  Call Extruder(256.15201)
  MoveL 1325 to (239.22, 155.88, 31.63) mm, rotated rx -180 ry 0 rz 180 deg; joints [-63.058, 52.64, -67.408, 63.827, 96.632, 13.225]
  MoveL 1326 to (239.22, 155.88, 31.63) mm, rotated rx -180 ry 0 rz 180 deg; joints [-63.058, 52.64, -67.408, 63.827, 96.632, 13.225]
  Call Extruder(256.33510)
  MoveL 1327 to (239.11, 156.17, 31.63) mm, rotated rx -180 ry 0 rz 180 deg; joints [-63.136, 52.655, -67.4, 63.902, 96.604, 13.213]
  MoveL 1328 to (239.11, 156.17, 31.63) mm, rotated rx -180 ry 0 rz 180 deg; joints [-63.136, 52.655, -67.4, 63.902, 96.604, 13.213]
  Call Extruder(256.49281)
  MoveL 1329 to (239, 156.42, 31.63) mm, rotated rx -180 ry 0 rz 180 deg; joints [-63.204, 52.668, -67.393, 63.966, 96.58, 13.203]
  MoveL 1330 to (239, 156.42, 31.63) mm, rotated rx -180 ry 0 rz 180 deg; joints [-63.204, 52.668, -67.393, 63.966, 96.58, 13.203]
  Call Extruder(256.65113)
  MoveL 1331 to (238.89, 156.67, 31.63) mm, rotated rx 180 ry 0 rz 180 deg; joints [-63.272, 52.68, -67.387, 64.031, 96.556, 13.193]
  MoveL 1332 to (238.89, 156.67, 31.63) mm, rotated rx 180 ry 0 rz 180 deg; joints [-63.272, 52.68, -67.387, 64.031, 96.556, 13.193]
  Call Extruder(256.83316)
  MoveL 1333 to (238.75, 156.94, 31.63) mm, rotated rx -180 ry 0 rz -180 deg; joints [-63.354, 52.694, -67.379, 64.109, 96.528, 13.183]
  MoveL 1334 to (238.75, 156.94, 31.63) mm, rotated rx -180 ry 0 rz -180 deg; joints [-63.354, 52.694, -67.379, 64.109, 96.528, 13.183]
  Call Extruder(257.03972)
  MoveL 1335 to (238.57, 157.25, 31.63) mm, rotated rx -180 ry 0 rz 180 deg; joints [-63.449, 52.708, -67.372, 64.2, 96.497, 13.174]
  MoveL 1336 to (238.57, 157.25, 31.63) mm, rotated rx -180 ry 0 rz 180 deg; joints [-63.449, 52.708, -67.372, 64.2, 96.497, 13.174]
  Call Extruder(257.24706)
  MoveL 1337 to (238.4, 157.55, 31.63) mm, rotated rx 180 ry 0 rz 180 deg; joints [-63.544, 52.722, -67.364, 64.291, 96.466, 13.165]
  MoveL 1338 to (238.4, 157.55, 31.63) mm, rotated rx 180 ry 0 rz 180 deg; joints [-63.544, 52.722, -67.364, 64.291, 96.466, 13.165]
  Call Extruder(257.45518)
  MoveL 1339 to (238.22, 157.85, 31.63) mm, rotated rx -180 ry 0 rz 180 deg; joints [-63.64, 52.736, -67.357, 64.383, 96.435, 13.156]
  MoveL 1340 to (238.22, 157.85, 31.63) mm, rotated rx -180 ry 0 rz 180 deg; joints [-63.64, 52.736, -67.357, 64.383, 96.435, 13.156]
  Call Extruder(257.57289)
  MoveL 1341 to (238.12, 158.02, 31.63) mm, rotated rx 180 ry 0 rz 180 deg; joints [-63.693, 52.744, -67.353, 64.434, 96.418, 13.151]
  MoveL 1342 to (238.12, 158.02, 31.63) mm, rotated rx 180 ry 0 rz 180 deg; joints [-63.693, 52.744, -67.353, 64.434, 96.418, 13.151]
  Call Extruder(257.90571)
  MoveL 1343 to (237.79, 158.48, 31.63) mm, rotated rx 180 ry 0 rz 180 deg; joints [-63.854, 52.763, -67.342, 64.588, 96.369, 13.142]
  MoveL 1344 to (237.79, 158.48, 31.63) mm, rotated rx 180 ry 0 rz 180 deg; joints [-63.854, 52.763, -67.342, 64.588, 96.369, 13.142]
  Call Extruder(258.23971)
  MoveL 1345 to (237.47, 158.93, 31.63) mm, rotated rx -180 ry 0 rz 180 deg; joints [-64.014, 52.782, -67.332, 64.742, 96.32, 13.133]
  MoveL 1346 to (237.47, 158.93, 31.63) mm, rotated rx -180 ry 0 rz 180 deg; joints [-64.014, 52.782, -67.332, 64.742, 96.32, 13.133]
  Call Extruder(258.40729)
  MoveL 1347 to (237.3, 159.15, 31.63) mm, rotated rx 180 ry 0 rz 180 deg; joints [-64.094, 52.792, -67.327, 64.819, 96.295, 13.128]
  Call Extruder(259.23663)
  MoveL 1348 to (236.39, 160.19, 31.63) mm, rotated rx -180 ry 0 rz 180 deg; joints [-64.505, 52.831, -67.306, 65.216, 96.177, 13.117]
  Call Extruder(259.86767)
  MoveL 1349 to (235.61, 160.89, 31.63) mm, rotated rx 180 ry 0 rz 180 deg; joints [-64.83, 52.852, -67.294, 65.531, 96.089, 13.121]
  MoveL 1350 to (235.61, 160.89, 31.63) mm, rotated rx 180 ry 0 rz 180 deg; joints [-64.83, 52.852, -67.294, 65.531, 96.089, 13.121]
  Call Extruder(260.06527)
  MoveL 1351 to (235.35, 161.1, 31.63) mm, rotated rx 180 ry 0 rz -180 deg; joints [-64.933, 52.858, -67.291, 65.631, 96.062, 13.123]
  Call Extruder(260.39930)
  MoveL 1352 to (234.9, 161.43, 31.63) mm, rotated rx -180 ry 0 rz -180 deg; joints [-65.109, 52.866, -67.287, 65.802, 96.017, 13.13]
  MoveL 1353 to (234.9, 161.43, 31.63) mm, rotated rx -180 ry 0 rz -180 deg; joints [-65.109, 52.866, -67.287, 65.802, 96.017, 13.13]
  Call Extruder(260.73214)
  MoveL 1354 to (234.45, 161.76, 31.63) mm, rotated rx -180 ry 0 rz -180 deg; joints [-65.285, 52.874, -67.282, 65.974, 95.972, 13.137]
  MoveL 1355 to (234.45, 161.76, 31.63) mm, rotated rx -180 ry 0 rz -180 deg; joints [-65.285, 52.874, -67.282, 65.974, 95.972, 13.137]
  Call Extruder(260.91134)
  MoveL 1356 to (234.21, 161.94, 31.63) mm, rotated rx 180 ry 0 rz -180 deg; joints [-65.381, 52.878, -67.28, 66.066, 95.947, 13.14]
  MoveL 1357 to (234.21, 161.94, 31.63) mm, rotated rx 180 ry 0 rz -180 deg; joints [-65.381, 52.878, -67.28, 66.066, 95.947, 13.14]
  Call Extruder(261.11946)
  MoveL 1358 to (233.9, 162.11, 31.63) mm, rotated rx 180 ry 0 rz -180 deg; joints [-65.493, 52.88, -67.279, 66.176, 95.92, 13.148]
  MoveL 1359 to (233.9, 162.11, 31.63) mm, rotated rx 180 ry 0 rz -180 deg; joints [-65.493, 52.88, -67.279, 66.176, 95.92, 13.148]
  Call Extruder(261.32679)
  MoveL 1360 to (233.6, 162.29, 31.63) mm, rotated rx -180 ry 0 rz 180 deg; joints [-65.605, 52.883, -67.277, 66.286, 95.893, 13.156]
  MoveL 1361 to (233.6, 162.29, 31.63) mm, rotated rx -180 ry 0 rz 180 deg; joints [-65.605, 52.883, -67.277, 66.286, 95.893, 13.156]
  Call Extruder(261.53335)
  MoveL 1362 to (233.29, 162.46, 31.63) mm, rotated rx 180 ry 0 rz 180 deg; joints [-65.718, 52.885, -67.276, 66.395, 95.866, 13.164]
  MoveL 1363 to (233.29, 162.46, 31.63) mm, rotated rx 180 ry 0 rz 180 deg; joints [-65.718, 52.885, -67.276, 66.395, 95.866, 13.164]
  Call Extruder(261.73913)
  MoveL 1364 to (232.99, 162.64, 31.63) mm, rotated rx -180 ry 0 rz 180 deg; joints [-65.83, 52.888, -67.275, 66.505, 95.839, 13.172]
  MoveL 1365 to (232.99, 162.64, 31.63) mm, rotated rx -180 ry 0 rz 180 deg; joints [-65.83, 52.888, -67.275, 66.505, 95.839, 13.172]
  Call Extruder(261.89741)
  MoveL 1366 to (232.74, 162.74, 31.63) mm, rotated rx -180 ry 0 rz 180 deg; joints [-65.917, 52.888, -67.275, 66.59, 95.819, 13.181]
  MoveL 1367 to (232.74, 162.74, 31.63) mm, rotated rx -180 ry 0 rz 180 deg; joints [-65.917, 52.888, -67.275, 66.59, 95.819, 13.181]
  Call Extruder(262.05508)
  MoveL 1368 to (232.49, 162.85, 31.63) mm, rotated rx -180 ry 0 rz 180 deg; joints [-66.004, 52.887, -67.275, 66.675, 95.8, 13.19]
  MoveL 1369 to (232.49, 162.85, 31.63) mm, rotated rx -180 ry 0 rz 180 deg; joints [-66.004, 52.887, -67.275, 66.675, 95.8, 13.19]
  Call Extruder(262.22517)
  MoveL 1370 to (232.22, 162.96, 31.63) mm, rotated rx 180 ry 0 rz 180 deg; joints [-66.099, 52.887, -67.275, 66.768, 95.778, 13.2]
  MoveL 1371 to (232.22, 162.96, 31.63) mm, rotated rx 180 ry 0 rz 180 deg; joints [-66.099, 52.887, -67.275, 66.768, 95.778, 13.2]
  Call Extruder(262.40753)
  MoveL 1372 to (231.93, 163.09, 31.63) mm, rotated rx -180 ry 0 rz 180 deg; joints [-66.2, 52.886, -67.275, 66.867, 95.755, 13.21]
  MoveL 1373 to (231.93, 163.09, 31.63) mm, rotated rx -180 ry 0 rz 180 deg; joints [-66.2, 52.886, -67.275, 66.867, 95.755, 13.21]
  Call Extruder(262.58914)
  MoveL 1374 to (231.64, 163.21, 31.63) mm, rotated rx -180 ry 0 rz 180 deg; joints [-66.302, 52.886, -67.276, 66.967, 95.733, 13.221]
  MoveL 1375 to (231.64, 163.21, 31.63) mm, rotated rx -180 ry 0 rz 180 deg; joints [-66.302, 52.886, -67.276, 66.967, 95.733, 13.221]
  Call Extruder(262.70258)
  MoveL 1376 to (231.45, 163.27, 31.63) mm, rotated rx -180 ry 0 rz -180 deg; joints [-66.365, 52.884, -67.277, 67.029, 95.719, 13.229]
  MoveL 1377 to (231.45, 163.27, 31.63) mm, rotated rx -180 ry 0 rz -180 deg; joints [-66.365, 52.884, -67.277, 67.029, 95.719, 13.229]
  Call Extruder(262.81558)
  MoveL 1378 to (231.26, 163.33, 31.63) mm, rotated rx 180 ry 0 rz -180 deg; joints [-66.428, 52.883, -67.277, 67.091, 95.705, 13.237]
  MoveL 1379 to (231.26, 163.33, 31.63) mm, rotated rx 180 ry 0 rz -180 deg; joints [-66.428, 52.883, -67.277, 67.091, 95.705, 13.237]
  Call Extruder(262.92814)
  MoveL 1380 to (231.07, 163.39, 31.63) mm, rotated rx 180 ry 0 rz 180 deg; joints [-66.492, 52.882, -67.278, 67.153, 95.692, 13.245]
  MoveL 1381 to (231.07, 163.39, 31.63) mm, rotated rx 180 ry 0 rz 180 deg; joints [-66.492, 52.882, -67.278, 67.153, 95.692, 13.245]
  Call Extruder(263.04025)
  MoveL 1382 to (230.88, 163.45, 31.63) mm, rotated rx 180 ry 0 rz 180 deg; joints [-66.555, 52.88, -67.279, 67.216, 95.678, 13.254]
  MoveL 1383 to (230.88, 163.45, 31.63) mm, rotated rx 180 ry 0 rz 180 deg; joints [-66.555, 52.88, -67.279, 67.216, 95.678, 13.254]
  Call Extruder(263.15191)
  MoveL 1384 to (230.69, 163.51, 31.63) mm, rotated rx 180 ry 0 rz -180 deg; joints [-66.619, 52.879, -67.28, 67.278, 95.664, 13.262]
  MoveL 1385 to (230.69, 163.51, 31.63) mm, rotated rx 180 ry 0 rz -180 deg; joints [-66.619, 52.879, -67.28, 67.278, 95.664, 13.262]
  Call Extruder(263.28301)
  MoveL 1386 to (230.47, 163.58, 31.63) mm, rotated rx -180 ry 0 rz 180 deg; joints [-66.694, 52.877, -67.281, 67.351, 95.648, 13.272]
  MoveL 1387 to (230.47, 163.58, 31.63) mm, rotated rx -180 ry 0 rz 180 deg; joints [-66.694, 52.877, -67.281, 67.351, 95.648, 13.272]
  Call Extruder(263.41354)
  MoveL 1388 to (230.25, 163.65, 31.63) mm, rotated rx -180 ry 0 rz 180 deg; joints [-66.768, 52.875, -67.282, 67.424, 95.632, 13.282]
  MoveL 1389 to (230.25, 163.65, 31.63) mm, rotated rx -180 ry 0 rz 180 deg; joints [-66.768, 52.875, -67.282, 67.424, 95.632, 13.282]
  Call Extruder(263.54350)
  MoveL 1390 to (230.02, 163.72, 31.63) mm, rotated rx 180 ry 0 rz -180 deg; joints [-66.843, 52.873, -67.283, 67.498, 95.616, 13.291]
  MoveL 1391 to (230.02, 163.72, 31.63) mm, rotated rx 180 ry 0 rz -180 deg; joints [-66.843, 52.873, -67.283, 67.498, 95.616, 13.291]
  Call Extruder(263.67290)
  MoveL 1392 to (229.8, 163.78, 31.63) mm, rotated rx 180 ry 0 rz -180 deg; joints [-66.918, 52.871, -67.284, 67.571, 95.6, 13.301]
  MoveL 1393 to (229.8, 163.78, 31.63) mm, rotated rx 180 ry 0 rz -180 deg; joints [-66.918, 52.871, -67.284, 67.571, 95.6, 13.301]
  Call Extruder(263.79488)
  MoveL 1394 to (229.59, 163.84, 31.63) mm, rotated rx -180 ry 0 rz 180 deg; joints [-66.988, 52.869, -67.285, 67.64, 95.585, 13.311]
  MoveL 1395 to (229.59, 163.84, 31.63) mm, rotated rx -180 ry 0 rz 180 deg; joints [-66.988, 52.869, -67.285, 67.64, 95.585, 13.311]
  Call Extruder(263.90973)
  MoveL 1396 to (229.38, 163.88, 31.63) mm, rotated rx 180 ry 0 rz 180 deg; joints [-67.054, 52.866, -67.287, 67.705, 95.572, 13.322]
  MoveL 1397 to (229.38, 163.88, 31.63) mm, rotated rx 180 ry 0 rz 180 deg; joints [-67.054, 52.866, -67.287, 67.705, 95.572, 13.322]
  Call Extruder(264.02412)
  MoveL 1398 to (229.18, 163.93, 31.63) mm, rotated rx 180 ry 0 rz -180 deg; joints [-67.12, 52.864, -67.288, 67.77, 95.558, 13.332]
  MoveL 1399 to (229.18, 163.93, 31.63) mm, rotated rx 180 ry 0 rz -180 deg; joints [-67.12, 52.864, -67.288, 67.77, 95.558, 13.332]
  Call Extruder(264.13806)
  MoveL 1400 to (228.97, 163.97, 31.63) mm, rotated rx -180 ry 0 rz 180 deg; joints [-67.187, 52.861, -67.29, 67.836, 95.544, 13.342]
  MoveL 1401 to (228.97, 163.97, 31.63) mm, rotated rx -180 ry 0 rz 180 deg; joints [-67.187, 52.861, -67.29, 67.836, 95.544, 13.342]
  Call Extruder(264.25155)
  MoveL 1402 to (228.77, 164.02, 31.63) mm, rotated rx 180 ry 0 rz 180 deg; joints [-67.253, 52.858, -67.291, 67.901, 95.531, 13.352]
  MoveL 1403 to (228.77, 164.02, 31.63) mm, rotated rx 180 ry 0 rz 180 deg; joints [-67.253, 52.858, -67.291, 67.901, 95.531, 13.352]
  Call Extruder(264.38884)
  MoveL 1404 to (228.52, 164.07, 31.63) mm, rotated rx 180 ry 0 rz 180 deg; joints [-67.333, 52.854, -67.293, 67.98, 95.514, 13.365]
  MoveL 1405 to (228.52, 164.07, 31.63) mm, rotated rx 180 ry 0 rz 180 deg; joints [-67.333, 52.854, -67.293, 67.98, 95.514, 13.365]
  Call Extruder(264.52551)
  MoveL 1406 to (228.27, 164.12, 31.63) mm, rotated rx 180 ry 0 rz -180 deg; joints [-67.413, 52.851, -67.295, 68.058, 95.498, 13.378]
  MoveL 1407 to (228.27, 164.12, 31.63) mm, rotated rx 180 ry 0 rz -180 deg; joints [-67.413, 52.851, -67.295, 68.058, 95.498, 13.378]
  Call Extruder(264.66157)
  MoveL 1408 to (228.02, 164.17, 31.63) mm, rotated rx 180 ry 0 rz 180 deg; joints [-67.494, 52.847, -67.297, 68.137, 95.481, 13.39]
  MoveL 1409 to (228.02, 164.17, 31.63) mm, rotated rx 180 ry 0 rz 180 deg; joints [-67.494, 52.847, -67.297, 68.137, 95.481, 13.39]
  Call Extruder(264.79703)
  MoveL 1410 to (227.77, 164.22, 31.63) mm, rotated rx 180 ry 0 rz -180 deg; joints [-67.574, 52.844, -67.299, 68.216, 95.465, 13.403]
  MoveL 1411 to (227.77, 164.22, 31.63) mm, rotated rx 180 ry 0 rz -180 deg; joints [-67.574, 52.844, -67.299, 68.216, 95.465, 13.403]
  Call Extruder(264.93187)
  MoveL 1412 to (227.52, 164.27, 31.63) mm, rotated rx -180 ry 0 rz -180 deg; joints [-67.654, 52.84, -67.301, 68.295, 95.448, 13.416]
  MoveL 1413 to (227.52, 164.27, 31.63) mm, rotated rx -180 ry 0 rz -180 deg; joints [-67.654, 52.84, -67.301, 68.295, 95.448, 13.416]
  Call Extruder(265.06610)
  MoveL 1414 to (227.27, 164.32, 31.63) mm, rotated rx 180 ry 0 rz -180 deg; joints [-67.735, 52.837, -67.303, 68.374, 95.431, 13.428]
  MoveL 1415 to (227.27, 164.32, 31.63) mm, rotated rx 180 ry 0 rz -180 deg; joints [-67.735, 52.837, -67.303, 68.374, 95.431, 13.428]
  Call Extruder(265.19972)
  MoveL 1416 to (227.03, 164.36, 31.63) mm, rotated rx -180 ry 0 rz 180 deg; joints [-67.815, 52.833, -67.305, 68.454, 95.415, 13.441]
  MoveL 1417 to (227.03, 164.36, 31.63) mm, rotated rx -180 ry 0 rz 180 deg; joints [-67.815, 52.833, -67.305, 68.454, 95.415, 13.441]
  Call Extruder(265.36183)
  MoveL 1418 to (226.72, 164.41, 31.63) mm, rotated rx -180 ry 0 rz 180 deg; joints [-67.912, 52.828, -67.307, 68.549, 95.395, 13.457]
  MoveL 1419 to (226.72, 164.41, 31.63) mm, rotated rx -180 ry 0 rz 180 deg; joints [-67.912, 52.828, -67.307, 68.549, 95.395, 13.457]
  Call Extruder(265.52320)
  MoveL 1420 to (226.41, 164.46, 31.63) mm, rotated rx -180 ry 0 rz 180 deg; joints [-68.01, 52.823, -67.31, 68.645, 95.375, 13.473]
  MoveL 1421 to (226.41, 164.46, 31.63) mm, rotated rx -180 ry 0 rz 180 deg; joints [-68.01, 52.823, -67.31, 68.645, 95.375, 13.473]
  Call Extruder(265.68385)
  MoveL 1422 to (226.11, 164.51, 31.63) mm, rotated rx -180 ry 0 rz -180 deg; joints [-68.107, 52.818, -67.313, 68.741, 95.355, 13.489]
  MoveL 1423 to (226.11, 164.51, 31.63) mm, rotated rx -180 ry 0 rz -180 deg; joints [-68.107, 52.818, -67.313, 68.741, 95.355, 13.489]
  Call Extruder(265.84377)
  MoveL 1424 to (225.8, 164.56, 31.63) mm, rotated rx -180 ry 0 rz -180 deg; joints [-68.205, 52.813, -67.316, 68.837, 95.335, 13.505]
  MoveL 1425 to (225.8, 164.56, 31.63) mm, rotated rx -180 ry 0 rz -180 deg; joints [-68.205, 52.813, -67.316, 68.837, 95.335, 13.505]
  Call Extruder(266.00296)
  MoveL 1426 to (225.5, 164.61, 31.63) mm, rotated rx -180 ry 0 rz -180 deg; joints [-68.303, 52.808, -67.318, 68.933, 95.315, 13.521]
  MoveL 1427 to (225.5, 164.61, 31.63) mm, rotated rx -180 ry 0 rz -180 deg; joints [-68.303, 52.808, -67.318, 68.933, 95.315, 13.521]
  Call Extruder(266.16143)
  MoveL 1428 to (225.19, 164.66, 31.63) mm, rotated rx -180 ry 0 rz 180 deg; joints [-68.4, 52.803, -67.321, 69.029, 95.295, 13.537]
  MoveL 1429 to (225.19, 164.66, 31.63) mm, rotated rx -180 ry 0 rz 180 deg; joints [-68.4, 52.803, -67.321, 69.029, 95.295, 13.537]
  Call Extruder(266.36030)
  MoveL 1430 to (224.8, 164.7, 31.63) mm, rotated rx -180 ry 0 rz 180 deg; joints [-68.522, 52.796, -67.325, 69.149, 95.27, 13.559]
  MoveL 1431 to (224.8, 164.7, 31.63) mm, rotated rx -180 ry 0 rz 180 deg; joints [-68.522, 52.796, -67.325, 69.149, 95.27, 13.559]
  Call Extruder(266.55831)
  MoveL 1432 to (224.42, 164.75, 31.63) mm, rotated rx 180 ry 0 rz 180 deg; joints [-68.645, 52.789, -67.329, 69.27, 95.245, 13.58]
  MoveL 1433 to (224.42, 164.75, 31.63) mm, rotated rx 180 ry 0 rz 180 deg; joints [-68.645, 52.789, -67.329, 69.27, 95.245, 13.58]
  Call Extruder(266.75545)
  MoveL 1434 to (224.03, 164.79, 31.63) mm, rotated rx 180 ry 0 rz 180 deg; joints [-68.767, 52.782, -67.333, 69.39, 95.221, 13.601]
  MoveL 1435 to (224.03, 164.79, 31.63) mm, rotated rx 180 ry 0 rz 180 deg; joints [-68.767, 52.782, -67.333, 69.39, 95.221, 13.601]
  Call Extruder(266.95173)
  MoveL 1436 to (223.64, 164.84, 31.63) mm, rotated rx 180 ry 0 rz -180 deg; joints [-68.89, 52.774, -67.336, 69.511, 95.196, 13.622]
  MoveL 1437 to (223.64, 164.84, 31.63) mm, rotated rx 180 ry 0 rz -180 deg; joints [-68.89, 52.774, -67.336, 69.511, 95.196, 13.622]
  Call Extruder(267.19740)
  MoveL 1438 to (223.15, 164.89, 31.63) mm, rotated rx 180 ry 0 rz 180 deg; joints [-69.043, 52.765, -67.342, 69.661, 95.165, 13.65]
  MoveL 1439 to (223.15, 164.89, 31.63) mm, rotated rx 180 ry 0 rz 180 deg; joints [-69.043, 52.765, -67.342, 69.661, 95.165, 13.65]
  Call Extruder(267.49209)
  MoveL 1440 to (222.56, 164.93, 31.63) mm, rotated rx 180 ry 0 rz 180 deg; joints [-69.227, 52.753, -67.348, 69.843, 95.128, 13.683]
  MoveL 1441 to (222.56, 164.93, 31.63) mm, rotated rx 180 ry 0 rz 180 deg; joints [-69.227, 52.753, -67.348, 69.843, 95.128, 13.683]
  Call Extruder(267.78545)
  MoveL 1442 to (221.97, 164.98, 31.63) mm, rotated rx 180 ry 0 rz 180 deg; joints [-69.411, 52.741, -67.354, 70.024, 95.09, 13.717]
  MoveL 1443 to (221.97, 164.98, 31.63) mm, rotated rx 180 ry 0 rz 180 deg; joints [-69.411, 52.741, -67.354, 70.024, 95.09, 13.717]
  Call Extruder(268.21876)
  MoveL 1444 to (221.1, 165.03, 31.63) mm, rotated rx 180 ry 0 rz -180 deg; joints [-69.684, 52.722, -67.365, 70.292, 95.035, 13.768]
  MoveL 1445 to (221.1, 165.03, 31.63) mm, rotated rx 180 ry 0 rz -180 deg; joints [-69.684, 52.722, -67.365, 70.292, 95.035, 13.768]
  Call Extruder(268.79092)
  MoveL 1446 to (219.94, 165.07, 31.63) mm, rotated rx -180 ry 0 rz 180 deg; joints [-70.044, 52.696, -67.379, 70.647, 94.963, 13.836]
  MoveL 1447 to (219.94, 165.07, 31.63) mm, rotated rx -180 ry 0 rz 180 deg; joints [-70.044, 52.696, -67.379, 70.647, 94.963, 13.836]
  Call Extruder(269.21879)
  MoveL 1448 to (219.06, 165.09, 31.63) mm, rotated rx -180 ry 0 rz 180 deg; joints [-70.315, 52.675, -67.389, 70.913, 94.908, 13.888]
  Call Extruder(385.86744)
  MoveL 1449 to (-19.06, 165.09, 31.63) mm, rotated rx -180 ry 0 rz 180 deg; joints [-137.325, 57.005, -63.843, 137.121, 84.978, 4.647]
  MoveL 1450 to (-19.06, 165.09, 31.63) mm, rotated rx -180 ry 0 rz 180 deg; joints [-137.325, 57.005, -63.843, 137.121, 84.978, 4.647]
  Call Extruder(386.58306)
  MoveL 1451 to (-20.52, 165.05, 31.63) mm, rotated rx 180 ry 0 rz -180 deg; joints [-137.563, 57.061, -63.774, 137.367, 85.05, 4.541]
  MoveL 1452 to (-20.52, 165.05, 31.63) mm, rotated rx 180 ry 0 rz -180 deg; joints [-137.563, 57.061, -63.774, 137.367, 85.05, 4.541]
  Call Extruder(387.15780)
  MoveL 1453 to (-21.68, 165, 31.63) mm, rotated rx -180 ry 0 rz -180 deg; joints [-137.754, 57.105, -63.719, 137.564, 85.108, 4.458]
  MoveL 1454 to (-21.68, 165, 31.63) mm, rotated rx -180 ry 0 rz -180 deg; joints [-137.754, 57.105, -63.719, 137.564, 85.108, 4.458]
  Call Extruder(387.45117)
  MoveL 1455 to (-22.27, 164.95, 31.63) mm, rotated rx 180 ry 0 rz 180 deg; joints [-137.855, 57.126, -63.692, 137.667, 85.136, 4.417]
  MoveL 1456 to (-22.27, 164.95, 31.63) mm, rotated rx 180 ry 0 rz 180 deg; joints [-137.855, 57.126, -63.692, 137.667, 85.136, 4.417]
  Call Extruder(387.74586)
  MoveL 1457 to (-22.86, 164.91, 31.63) mm, rotated rx 180 ry 0 rz -180 deg; joints [-137.955, 57.148, -63.665, 137.77, 85.165, 4.375]
  MoveL 1458 to (-22.86, 164.91, 31.63) mm, rotated rx 180 ry 0 rz -180 deg; joints [-137.955, 57.148, -63.665, 137.77, 85.165, 4.375]
  Call Extruder(388.04189)
  MoveL 1459 to (-23.45, 164.86, 31.63) mm, rotated rx -180 ry 0 rz -180 deg; joints [-138.054, 57.169, -63.638, 137.872, 85.193, 4.334]
  MoveL 1460 to (-23.45, 164.86, 31.63) mm, rotated rx -180 ry 0 rz -180 deg; joints [-138.054, 57.169, -63.638, 137.872, 85.193, 4.334]
  Call Extruder(388.23816)
  MoveL 1461 to (-23.83, 164.82, 31.63) mm, rotated rx -180 ry 0 rz 180 deg; joints [-138.122, 57.183, -63.621, 137.942, 85.211, 4.308]
  MoveL 1462 to (-23.83, 164.82, 31.63) mm, rotated rx -180 ry 0 rz 180 deg; joints [-138.122, 57.183, -63.621, 137.942, 85.211, 4.308]
  Call Extruder(388.43530)
  MoveL 1463 to (-24.22, 164.77, 31.63) mm, rotated rx 180 ry 0 rz 180 deg; joints [-138.19, 57.196, -63.604, 138.012, 85.229, 4.282]
  MoveL 1464 to (-24.22, 164.77, 31.63) mm, rotated rx 180 ry 0 rz 180 deg; joints [-138.19, 57.196, -63.604, 138.012, 85.229, 4.282]
  Call Extruder(388.63331)
  MoveL 1465 to (-24.61, 164.72, 31.63) mm, rotated rx -180 ry 0 rz -180 deg; joints [-138.258, 57.21, -63.586, 138.081, 85.246, 4.255]
  MoveL 1466 to (-24.61, 164.72, 31.63) mm, rotated rx -180 ry 0 rz -180 deg; joints [-138.258, 57.21, -63.586, 138.081, 85.246, 4.255]
  Call Extruder(388.83219)
  MoveL 1467 to (-25, 164.68, 31.63) mm, rotated rx -180 ry 0 rz 180 deg; joints [-138.325, 57.223, -63.569, 138.151, 85.265, 4.229]
  MoveL 1468 to (-25, 164.68, 31.63) mm, rotated rx -180 ry 0 rz 180 deg; joints [-138.325, 57.223, -63.569, 138.151, 85.265, 4.229]
  Call Extruder(389.01127)
  MoveL 1469 to (-25.34, 164.63, 31.63) mm, rotated rx 180 ry 0 rz 180 deg; joints [-138.387, 57.235, -63.554, 138.213, 85.28, 4.206]
  MoveL 1470 to (-25.34, 164.63, 31.63) mm, rotated rx 180 ry 0 rz 180 deg; joints [-138.387, 57.235, -63.554, 138.213, 85.28, 4.206]
  Call Extruder(389.17046)
  MoveL 1471 to (-25.65, 164.58, 31.63) mm, rotated rx -180 ry 0 rz 180 deg; joints [-138.442, 57.245, -63.54, 138.27, 85.294, 4.185]
  MoveL 1472 to (-25.65, 164.58, 31.63) mm, rotated rx -180 ry 0 rz 180 deg; joints [-138.442, 57.245, -63.54, 138.27, 85.294, 4.185]
  Call Extruder(389.33039)
  MoveL 1473 to (-25.96, 164.54, 31.63) mm, rotated rx 180 ry 0 rz -180 deg; joints [-138.497, 57.256, -63.527, 138.327, 85.307, 4.165]
  MoveL 1474 to (-25.96, 164.54, 31.63) mm, rotated rx 180 ry 0 rz -180 deg; joints [-138.497, 57.256, -63.527, 138.327, 85.307, 4.165]
  Call Extruder(389.49104)
  MoveL 1475 to (-26.26, 164.49, 31.63) mm, rotated rx 180 ry 0 rz 180 deg; joints [-138.552, 57.266, -63.514, 138.383, 85.321, 4.145]
  MoveL 1476 to (-26.26, 164.49, 31.63) mm, rotated rx 180 ry 0 rz 180 deg; joints [-138.552, 57.266, -63.514, 138.383, 85.321, 4.145]
  Call Extruder(389.65242)
  MoveL 1477 to (-26.57, 164.44, 31.63) mm, rotated rx -180 ry 0 rz 180 deg; joints [-138.607, 57.276, -63.5, 138.439, 85.335, 4.125]
  MoveL 1478 to (-26.57, 164.44, 31.63) mm, rotated rx -180 ry 0 rz 180 deg; joints [-138.607, 57.276, -63.5, 138.439, 85.335, 4.125]
  Call Extruder(389.81452)
  MoveL 1479 to (-26.87, 164.39, 31.63) mm, rotated rx -180 ry 0 rz 180 deg; joints [-138.662, 57.287, -63.487, 138.496, 85.348, 4.104]
  MoveL 1480 to (-26.87, 164.39, 31.63) mm, rotated rx -180 ry 0 rz 180 deg; joints [-138.662, 57.287, -63.487, 138.496, 85.348, 4.104]
  Call Extruder(389.96273)
  MoveL 1481 to (-27.15, 164.34, 31.63) mm, rotated rx 180 ry 0 rz -180 deg; joints [-138.713, 57.296, -63.475, 138.547, 85.361, 4.086]
  MoveL 1482 to (-27.15, 164.34, 31.63) mm, rotated rx 180 ry 0 rz -180 deg; joints [-138.713, 57.296, -63.475, 138.547, 85.361, 4.086]
  Call Extruder(390.09696)
  MoveL 1483 to (-27.4, 164.29, 31.63) mm, rotated rx -180 ry 0 rz 180 deg; joints [-138.759, 57.304, -63.465, 138.595, 85.371, 4.07]
  MoveL 1484 to (-27.4, 164.29, 31.63) mm, rotated rx -180 ry 0 rz 180 deg; joints [-138.759, 57.304, -63.465, 138.595, 85.371, 4.07]
  Call Extruder(390.23180)
  MoveL 1485 to (-27.65, 164.24, 31.63) mm, rotated rx -180 ry 0 rz 180 deg; joints [-138.806, 57.312, -63.454, 138.642, 85.382, 4.054]
  MoveL 1486 to (-27.65, 164.24, 31.63) mm, rotated rx -180 ry 0 rz 180 deg; joints [-138.806, 57.312, -63.454, 138.642, 85.382, 4.054]
  Call Extruder(390.36725)
  MoveL 1487 to (-27.9, 164.19, 31.63) mm, rotated rx -180 ry 0 rz 180 deg; joints [-138.852, 57.32, -63.444, 138.689, 85.392, 4.038]
  MoveL 1488 to (-27.9, 164.19, 31.63) mm, rotated rx -180 ry 0 rz 180 deg; joints [-138.852, 57.32, -63.444, 138.689, 85.392, 4.038]
  Call Extruder(390.50331)
  MoveL 1489 to (-28.15, 164.14, 31.63) mm, rotated rx -180 ry 0 rz 180 deg; joints [-138.898, 57.328, -63.433, 138.736, 85.403, 4.022]
  MoveL 1490 to (-28.15, 164.14, 31.63) mm, rotated rx -180 ry 0 rz 180 deg; joints [-138.898, 57.328, -63.433, 138.736, 85.403, 4.022]
  Call Extruder(390.63999)
  MoveL 1491 to (-28.4, 164.09, 31.63) mm, rotated rx 180 ry 0 rz 180 deg; joints [-138.944, 57.336, -63.422, 138.784, 85.414, 4.006]
  MoveL 1492 to (-28.4, 164.09, 31.63) mm, rotated rx 180 ry 0 rz 180 deg; joints [-138.944, 57.336, -63.422, 138.784, 85.414, 4.006]
  Call Extruder(390.77727)
  MoveL 1493 to (-28.65, 164.04, 31.63) mm, rotated rx -180 ry 0 rz 180 deg; joints [-138.99, 57.344, -63.412, 138.831, 85.425, 3.99]
  MoveL 1494 to (-28.65, 164.04, 31.63) mm, rotated rx -180 ry 0 rz 180 deg; joints [-138.99, 57.344, -63.412, 138.831, 85.425, 3.99]
  Call Extruder(390.90294)
  MoveL 1495 to (-28.87, 164, 31.63) mm, rotated rx -180 ry 0 rz -180 deg; joints [-139.032, 57.351, -63.402, 138.874, 85.434, 3.976]
  MoveL 1496 to (-28.87, 164, 31.63) mm, rotated rx -180 ry 0 rz -180 deg; joints [-139.032, 57.351, -63.402, 138.874, 85.434, 3.976]
  Call Extruder(391.01688)
  MoveL 1497 to (-29.08, 163.95, 31.63) mm, rotated rx -180 ry 0 rz 180 deg; joints [-139.071, 57.357, -63.394, 138.913, 85.443, 3.963]
  MoveL 1498 to (-29.08, 163.95, 31.63) mm, rotated rx -180 ry 0 rz 180 deg; joints [-139.071, 57.357, -63.394, 138.913, 85.443, 3.963]
  Call Extruder(391.13127)
  MoveL 1499 to (-29.28, 163.91, 31.63) mm, rotated rx -180 ry 0 rz -180 deg; joints [-139.109, 57.364, -63.385, 138.952, 85.452, 3.95]
  MoveL 1500 to (-29.28, 163.91, 31.63) mm, rotated rx -180 ry 0 rz -180 deg; joints [-139.109, 57.364, -63.385, 138.952, 85.452, 3.95]
  Call Extruder(391.24612)
  MoveL 1501 to (-29.48, 163.86, 31.63) mm, rotated rx 180 ry 0 rz 180 deg; joints [-139.147, 57.37, -63.377, 138.991, 85.46, 3.937]
  MoveL 1502 to (-29.48, 163.86, 31.63) mm, rotated rx 180 ry 0 rz 180 deg; joints [-139.147, 57.37, -63.377, 138.991, 85.46, 3.937]
  Call Extruder(391.36141)
  MoveL 1503 to (-29.69, 163.82, 31.63) mm, rotated rx -180 ry 0 rz -180 deg; joints [-139.186, 57.377, -63.368, 139.03, 85.469, 3.924]
  MoveL 1504 to (-29.69, 163.82, 31.63) mm, rotated rx -180 ry 0 rz -180 deg; joints [-139.186, 57.377, -63.368, 139.03, 85.469, 3.924]
  Call Extruder(391.49081)
  MoveL 1505 to (-29.91, 163.75, 31.63) mm, rotated rx -180 ry 0 rz -180 deg; joints [-139.231, 57.383, -63.359, 139.076, 85.477, 3.911]
  MoveL 1506 to (-29.91, 163.75, 31.63) mm, rotated rx -180 ry 0 rz -180 deg; joints [-139.231, 57.383, -63.359, 139.076, 85.477, 3.911]
  Call Extruder(391.62077)
  MoveL 1507 to (-30.14, 163.68, 31.63) mm, rotated rx 180 ry 0 rz 180 deg; joints [-139.276, 57.39, -63.351, 139.122, 85.486, 3.897]
  MoveL 1508 to (-30.14, 163.68, 31.63) mm, rotated rx 180 ry 0 rz 180 deg; joints [-139.276, 57.39, -63.351, 139.122, 85.486, 3.897]
  Call Extruder(391.75130)
  MoveL 1509 to (-30.36, 163.61, 31.63) mm, rotated rx -180 ry 0 rz 180 deg; joints [-139.321, 57.396, -63.342, 139.168, 85.494, 3.884]
  MoveL 1510 to (-30.36, 163.61, 31.63) mm, rotated rx -180 ry 0 rz 180 deg; joints [-139.321, 57.396, -63.342, 139.168, 85.494, 3.884]
  Call Extruder(391.88239)
  MoveL 1511 to (-30.58, 163.55, 31.63) mm, rotated rx -180 ry 0 rz 180 deg; joints [-139.366, 57.403, -63.334, 139.214, 85.502, 3.87]
  MoveL 1512 to (-30.58, 163.55, 31.63) mm, rotated rx -180 ry 0 rz 180 deg; joints [-139.366, 57.403, -63.334, 139.214, 85.502, 3.87]
  Call Extruder(392.00403)
  MoveL 1513 to (-30.79, 163.48, 31.63) mm, rotated rx -180 ry 0 rz 180 deg; joints [-139.408, 57.408, -63.326, 139.256, 85.51, 3.858]
  MoveL 1514 to (-30.79, 163.48, 31.63) mm, rotated rx -180 ry 0 rz 180 deg; joints [-139.408, 57.408, -63.326, 139.256, 85.51, 3.858]
  Call Extruder(392.11615)
  MoveL 1515 to (-30.98, 163.42, 31.63) mm, rotated rx -180 ry 0 rz -180 deg; joints [-139.446, 57.414, -63.319, 139.295, 85.517, 3.847]
  MoveL 1516 to (-30.98, 163.42, 31.63) mm, rotated rx -180 ry 0 rz -180 deg; joints [-139.446, 57.414, -63.319, 139.295, 85.517, 3.847]
  Call Extruder(392.22871)
  MoveL 1517 to (-31.17, 163.36, 31.63) mm, rotated rx -180 ry 0 rz -180 deg; joints [-139.485, 57.419, -63.311, 139.335, 85.524, 3.836]
  MoveL 1518 to (-31.17, 163.36, 31.63) mm, rotated rx -180 ry 0 rz -180 deg; joints [-139.485, 57.419, -63.311, 139.335, 85.524, 3.836]
  Call Extruder(392.34171)
  MoveL 1519 to (-31.35, 163.3, 31.63) mm, rotated rx -180 ry 0 rz 180 deg; joints [-139.523, 57.424, -63.304, 139.374, 85.531, 3.825]
  MoveL 1520 to (-31.35, 163.3, 31.63) mm, rotated rx -180 ry 0 rz 180 deg; joints [-139.523, 57.424, -63.304, 139.374, 85.531, 3.825]
  Call Extruder(392.45516)
  MoveL 1521 to (-31.54, 163.24, 31.63) mm, rotated rx 180 ry 0 rz -180 deg; joints [-139.562, 57.43, -63.297, 139.413, 85.537, 3.814]
  MoveL 1522 to (-31.54, 163.24, 31.63) mm, rotated rx 180 ry 0 rz -180 deg; joints [-139.562, 57.43, -63.297, 139.413, 85.537, 3.814]
  Call Extruder(392.60280)
  MoveL 1523 to (-31.78, 163.15, 31.63) mm, rotated rx -180 ry 0 rz 180 deg; joints [-139.613, 57.436, -63.289, 139.465, 85.545, 3.8]
  MoveL 1524 to (-31.78, 163.15, 31.63) mm, rotated rx -180 ry 0 rz 180 deg; joints [-139.613, 57.436, -63.289, 139.465, 85.545, 3.8]
  Call Extruder(392.78516)
  MoveL 1525 to (-32.08, 163.02, 31.63) mm, rotated rx 180 ry 0 rz 180 deg; joints [-139.677, 57.443, -63.279, 139.53, 85.554, 3.784]
  MoveL 1526 to (-32.08, 163.02, 31.63) mm, rotated rx 180 ry 0 rz 180 deg; joints [-139.677, 57.443, -63.279, 139.53, 85.554, 3.784]
  Call Extruder(392.96827)
  MoveL 1527 to (-32.37, 162.91, 31.63) mm, rotated rx -180 ry 0 rz -180 deg; joints [-139.741, 57.451, -63.269, 139.595, 85.563, 3.767]
  MoveL 1528 to (-32.37, 162.91, 31.63) mm, rotated rx -180 ry 0 rz -180 deg; joints [-139.741, 57.451, -63.269, 139.595, 85.563, 3.767]
  Call Extruder(393.12594)
  MoveL 1529 to (-32.62, 162.8, 31.63) mm, rotated rx 180 ry 0 rz 180 deg; joints [-139.796, 57.457, -63.26, 139.65, 85.571, 3.754]
  MoveL 1530 to (-32.62, 162.8, 31.63) mm, rotated rx 180 ry 0 rz 180 deg; joints [-139.796, 57.457, -63.26, 139.65, 85.571, 3.754]
  Call Extruder(393.28422)
  MoveL 1531 to (-32.86, 162.69, 31.63) mm, rotated rx 180 ry 0 rz 180 deg; joints [-139.851, 57.463, -63.252, 139.706, 85.578, 3.74]
  MoveL 1532 to (-32.86, 162.69, 31.63) mm, rotated rx 180 ry 0 rz 180 deg; joints [-139.851, 57.463, -63.252, 139.706, 85.578, 3.74]
  Call Extruder(393.46623)
  MoveL 1533 to (-33.14, 162.55, 31.63) mm, rotated rx -180 ry 0 rz 180 deg; joints [-139.916, 57.469, -63.244, 139.772, 85.585, 3.726]
  MoveL 1534 to (-33.14, 162.55, 31.63) mm, rotated rx -180 ry 0 rz 180 deg; joints [-139.916, 57.469, -63.244, 139.772, 85.585, 3.726]
  Call Extruder(393.67279)
  MoveL 1535 to (-33.45, 162.37, 31.63) mm, rotated rx -180 ry 0 rz -180 deg; joints [-139.991, 57.475, -63.235, 139.848, 85.591, 3.711]
  MoveL 1536 to (-33.45, 162.37, 31.63) mm, rotated rx -180 ry 0 rz -180 deg; joints [-139.991, 57.475, -63.235, 139.848, 85.591, 3.711]
  Call Extruder(393.88012)
  MoveL 1537 to (-33.75, 162.2, 31.63) mm, rotated rx 180 ry 0 rz -180 deg; joints [-140.065, 57.481, -63.227, 139.923, 85.597, 3.695]
  MoveL 1538 to (-33.75, 162.2, 31.63) mm, rotated rx 180 ry 0 rz -180 deg; joints [-140.065, 57.481, -63.227, 139.923, 85.597, 3.695]
  Call Extruder(394.08824)
  MoveL 1539 to (-34.05, 162.02, 31.63) mm, rotated rx 180 ry 0 rz 180 deg; joints [-140.14, 57.487, -63.219, 139.999, 85.604, 3.68]
  MoveL 1540 to (-34.05, 162.02, 31.63) mm, rotated rx 180 ry 0 rz 180 deg; joints [-140.14, 57.487, -63.219, 139.999, 85.604, 3.68]
  Call Extruder(394.20594)
  MoveL 1541 to (-34.23, 161.92, 31.63) mm, rotated rx 180 ry 0 rz 180 deg; joints [-140.182, 57.491, -63.214, 140.041, 85.607, 3.672]
  MoveL 1542 to (-34.23, 161.92, 31.63) mm, rotated rx 180 ry 0 rz 180 deg; joints [-140.182, 57.491, -63.214, 140.041, 85.607, 3.672]
  Call Extruder(394.53878)
  MoveL 1543 to (-34.68, 161.59, 31.63) mm, rotated rx 180 ry 0 rz 180 deg; joints [-140.305, 57.498, -63.204, 140.165, 85.612, 3.652]
  MoveL 1544 to (-34.68, 161.59, 31.63) mm, rotated rx 180 ry 0 rz 180 deg; joints [-140.305, 57.498, -63.204, 140.165, 85.612, 3.652]
  Call Extruder(394.87281)
  MoveL 1545 to (-35.13, 161.27, 31.63) mm, rotated rx -180 ry 0 rz 180 deg; joints [-140.427, 57.505, -63.195, 140.288, 85.617, 3.632]
  MoveL 1546 to (-35.13, 161.27, 31.63) mm, rotated rx -180 ry 0 rz 180 deg; joints [-140.427, 57.505, -63.195, 140.288, 85.617, 3.632]
  Call Extruder(395.04040)
  MoveL 1547 to (-35.35, 161.1, 31.63) mm, rotated rx 180 ry 0 rz 180 deg; joints [-140.489, 57.508, -63.19, 140.35, 85.62, 3.622]
  Call Extruder(395.86969)
  MoveL 1548 to (-36.39, 160.19, 31.63) mm, rotated rx 180 ry 0 rz 180 deg; joints [-140.797, 57.52, -63.174, 140.66, 85.621, 3.581]
  Call Extruder(396.50077)
  MoveL 1549 to (-37.09, 159.4, 31.63) mm, rotated rx -180 ry 0 rz -180 deg; joints [-141.034, 57.522, -63.171, 140.898, 85.611, 3.559]
  MoveL 1550 to (-37.09, 159.4, 31.63) mm, rotated rx -180 ry 0 rz -180 deg; joints [-141.034, 57.522, -63.171, 140.898, 85.611, 3.559]
  Call Extruder(396.69836)
  MoveL 1551 to (-37.3, 159.15, 31.63) mm, rotated rx -180 ry 0 rz 180 deg; joints [-141.109, 57.522, -63.17, 140.972, 85.607, 3.553]
  Call Extruder(397.03238)
  MoveL 1552 to (-37.63, 158.7, 31.63) mm, rotated rx -180 ry 0 rz 180 deg; joints [-141.235, 57.521, -63.172, 141.098, 85.596, 3.546]
  MoveL 1553 to (-37.63, 158.7, 31.63) mm, rotated rx -180 ry 0 rz 180 deg; joints [-141.235, 57.521, -63.172, 141.098, 85.596, 3.546]
  Call Extruder(397.26956)
  MoveL 1554 to (-37.87, 158.38, 31.63) mm, rotated rx 180 ry 0 rz 180 deg; joints [-141.324, 57.52, -63.174, 141.188, 85.589, 3.54]
  Set speed (130.0 mm/s)
  MoveL 1555 to (-39.5, 155.42, 31.63) mm, rotated rx -180 ry 0 rz -180 deg; joints [-142.08, 57.492, -63.212, 141.941, 85.491, 3.522]
  MoveL 1556 to (-39.51, 155.42, 41.04) mm, rotated rx -180 ry 0 rz 180 deg; joints [-142.08, 58.93, -65.352, 141.905, 84.938, 3.957]
  Call Extruder(395.26956)
  Set speed (40.0 mm/s)
  MoveL 1557 to (-39.51, 155.42, 41.04) mm, rotated rx -180 ry 0 rz 180 deg; joints [-142.08, 58.93, -65.352, 141.905, 84.938, 3.957]
  Call Extruder(0.00000)
  Set speed (130.0 mm/s)
  MoveL 1558 to (-39.41, 155.44, 41.04) mm, rotated rx -180 ry 0 rz 180 deg; joints [-142.064, 58.926, -65.356, 141.888, 84.932, 3.964]
  Call Extruder(2.00000)
  Set speed (40.0 mm/s)
  MoveL 1559 to (-39.41, 155.44, 41.04) mm, rotated rx -180 ry 0 rz 180 deg; joints [-142.064, 58.926, -65.356, 141.888, 84.932, 3.964]
  Set speed (30.0 mm/s)
  MoveL 1560 to (-39.41, 155.44, 41.04) mm, rotated rx -180 ry 0 rz 180 deg; joints [-142.064, 58.926, -65.356, 141.888, 84.932, 3.964]
  Call Extruder(2.05684)
  MoveL 1561 to (-39.44, 155.34, 41.04) mm, rotated rx -180 ry 0 rz 180 deg; joints [-142.085, 58.924, -65.359, 141.909, 84.928, 3.964]
  MoveL 1562 to (-39.44, 155.34, 41.04) mm, rotated rx -180 ry 0 rz 180 deg; joints [-142.085, 58.924, -65.359, 141.909, 84.928, 3.964]
  Call Extruder(2.17007)
  MoveL 1563 to (-39.5, 155.15, 41.04) mm, rotated rx -180 ry 0 rz -180 deg; joints [-142.127, 58.921, -65.363, 141.951, 84.918, 3.966]
  MoveL 1564 to (-39.5, 155.15, 41.04) mm, rotated rx -180 ry 0 rz -180 deg; joints [-142.127, 58.921, -65.363, 141.951, 84.918, 3.966]
  Call Extruder(2.28286)
  MoveL 1565 to (-39.56, 154.97, 41.04) mm, rotated rx -180 ry 0 rz 180 deg; joints [-142.169, 58.917, -65.368, 141.993, 84.909, 3.967]
  MoveL 1566 to (-39.56, 154.97, 41.04) mm, rotated rx -180 ry 0 rz 180 deg; joints [-142.169, 58.917, -65.368, 141.993, 84.909, 3.967]
  Call Extruder(2.39521)
  MoveL 1567 to (-39.62, 154.78, 41.04) mm, rotated rx 180 ry 0 rz -180 deg; joints [-142.212, 58.914, -65.373, 142.035, 84.9, 3.968]
  MoveL 1568 to (-39.62, 154.78, 41.04) mm, rotated rx 180 ry 0 rz -180 deg; joints [-142.212, 58.914, -65.373, 142.035, 84.9, 3.968]
  Call Extruder(2.50711)
  MoveL 1569 to (-39.68, 154.59, 41.04) mm, rotated rx -180 ry 0 rz -180 deg; joints [-142.254, 58.91, -65.377, 142.077, 84.89, 3.969]
  MoveL 1570 to (-39.68, 154.59, 41.04) mm, rotated rx -180 ry 0 rz -180 deg; joints [-142.254, 58.91, -65.377, 142.077, 84.89, 3.969]
  Call Extruder(2.62851)
  MoveL 1571 to (-39.75, 154.38, 41.04) mm, rotated rx 180 ry 0 rz 180 deg; joints [-142.3, 58.906, -65.382, 142.122, 84.88, 3.971]
  MoveL 1572 to (-39.75, 154.38, 41.04) mm, rotated rx 180 ry 0 rz 180 deg; joints [-142.3, 58.906, -65.382, 142.122, 84.88, 3.971]
  Call Extruder(2.75930)
  MoveL 1573 to (-39.82, 154.16, 41.04) mm, rotated rx 180 ry 0 rz 180 deg; joints [-142.35, 58.902, -65.388, 142.171, 84.869, 3.973]
  MoveL 1574 to (-39.82, 154.16, 41.04) mm, rotated rx 180 ry 0 rz 180 deg; joints [-142.35, 58.902, -65.388, 142.171, 84.869, 3.973]
  Call Extruder(2.88953)
  MoveL 1575 to (-39.88, 153.94, 41.04) mm, rotated rx 180 ry 0 rz -180 deg; joints [-142.399, 58.898, -65.394, 142.22, 84.857, 3.974]
  MoveL 1576 to (-39.88, 153.94, 41.04) mm, rotated rx 180 ry 0 rz -180 deg; joints [-142.399, 58.898, -65.394, 142.22, 84.857, 3.974]
  Call Extruder(3.01920)
  MoveL 1577 to (-39.95, 153.71, 41.04) mm, rotated rx -180 ry 0 rz 180 deg; joints [-142.449, 58.893, -65.399, 142.27, 84.846, 3.976]
  MoveL 1578 to (-39.95, 153.71, 41.04) mm, rotated rx -180 ry 0 rz 180 deg; joints [-142.449, 58.893, -65.399, 142.27, 84.846, 3.976]
  Call Extruder(3.14830)
  MoveL 1579 to (-40.02, 153.49, 41.04) mm, rotated rx -180 ry 0 rz -180 deg; joints [-142.498, 58.889, -65.405, 142.319, 84.835, 3.978]
  MoveL 1580 to (-40.02, 153.49, 41.04) mm, rotated rx -180 ry 0 rz -180 deg; joints [-142.498, 58.889, -65.405, 142.319, 84.835, 3.978]
  Call Extruder(3.26338)
  MoveL 1581 to (-40.06, 153.28, 41.03) mm, rotated rx -180 ry 0 rz 180 deg; joints [-142.541, 58.884, -65.411, 142.361, 84.823, 3.98]
  MoveL 1582 to (-40.06, 153.28, 41.03) mm, rotated rx -180 ry 0 rz 180 deg; joints [-142.541, 58.884, -65.411, 142.361, 84.823, 3.98]
  Call Extruder(3.37802)
  MoveL 1583 to (-40.11, 153.08, 41.04) mm, rotated rx -180 ry 0 rz 180 deg; joints [-142.584, 58.88, -65.417, 142.404, 84.812, 3.983]
  MoveL 1584 to (-40.11, 153.08, 41.04) mm, rotated rx -180 ry 0 rz 180 deg; joints [-142.584, 58.88, -65.417, 142.404, 84.812, 3.983]
  Call Extruder(3.49220)
  MoveL 1585 to (-40.15, 152.88, 41.04) mm, rotated rx -180 ry 0 rz 180 deg; joints [-142.627, 58.875, -65.423, 142.446, 84.8, 3.986]
  MoveL 1586 to (-40.15, 152.88, 41.04) mm, rotated rx -180 ry 0 rz 180 deg; joints [-142.627, 58.875, -65.423, 142.446, 84.8, 3.986]
  Call Extruder(3.60593)
  MoveL 1587 to (-40.2, 152.67, 41.04) mm, rotated rx -180 ry 0 rz 180 deg; joints [-142.671, 58.87, -65.429, 142.489, 84.789, 3.988]
  MoveL 1588 to (-40.2, 152.67, 41.04) mm, rotated rx -180 ry 0 rz 180 deg; joints [-142.671, 58.87, -65.429, 142.489, 84.789, 3.988]
  Call Extruder(3.73136)
  MoveL 1589 to (-40.24, 152.45, 41.04) mm, rotated rx -180 ry 0 rz -180 deg; joints [-142.718, 58.865, -65.436, 142.536, 84.776, 3.991]
  MoveL 1590 to (-40.24, 152.45, 41.04) mm, rotated rx -180 ry 0 rz -180 deg; joints [-142.718, 58.865, -65.436, 142.536, 84.776, 3.991]
  Call Extruder(3.86834)
  MoveL 1591 to (-40.29, 152.2, 41.04) mm, rotated rx -180 ry 0 rz 180 deg; joints [-142.77, 58.859, -65.444, 142.587, 84.762, 3.995]
  MoveL 1592 to (-40.29, 152.2, 41.04) mm, rotated rx -180 ry 0 rz 180 deg; joints [-142.77, 58.859, -65.444, 142.587, 84.762, 3.995]
  Call Extruder(4.00470)
  MoveL 1593 to (-40.34, 151.95, 41.04) mm, rotated rx -180 ry 0 rz -180 deg; joints [-142.822, 58.853, -65.451, 142.639, 84.747, 3.998]
  MoveL 1594 to (-40.34, 151.95, 41.04) mm, rotated rx -180 ry 0 rz -180 deg; joints [-142.822, 58.853, -65.451, 142.639, 84.747, 3.998]
  Call Extruder(4.14046)
  MoveL 1595 to (-40.39, 151.7, 41.03) mm, rotated rx -180 ry 0 rz 180 deg; joints [-142.874, 58.848, -65.459, 142.69, 84.733, 4.002]
  MoveL 1596 to (-40.39, 151.7, 41.03) mm, rotated rx -180 ry 0 rz 180 deg; joints [-142.874, 58.848, -65.459, 142.69, 84.733, 4.002]
  Call Extruder(4.27560)
  MoveL 1597 to (-40.44, 151.45, 41.04) mm, rotated rx -180 ry 0 rz 180 deg; joints [-142.926, 58.842, -65.467, 142.741, 84.719, 4.005]
  MoveL 1598 to (-40.44, 151.45, 41.04) mm, rotated rx -180 ry 0 rz 180 deg; joints [-142.926, 58.842, -65.467, 142.741, 84.719, 4.005]
  Call Extruder(4.41014)
  MoveL 1599 to (-40.49, 151.2, 41.04) mm, rotated rx 180 ry 0 rz 180 deg; joints [-142.978, 58.836, -65.474, 142.793, 84.704, 4.008]
  MoveL 1600 to (-40.49, 151.2, 41.04) mm, rotated rx 180 ry 0 rz 180 deg; joints [-142.978, 58.836, -65.474, 142.793, 84.704, 4.008]
  Call Extruder(4.54406)
  MoveL 1601 to (-40.54, 150.95, 41.04) mm, rotated rx -180 ry 0 rz -180 deg; joints [-143.031, 58.83, -65.482, 142.844, 84.69, 4.012]
  MoveL 1602 to (-40.54, 150.95, 41.04) mm, rotated rx -180 ry 0 rz -180 deg; joints [-143.031, 58.83, -65.482, 142.844, 84.69, 4.012]
  Call Extruder(4.69192)
  MoveL 1603 to (-40.59, 150.67, 41.04) mm, rotated rx 180 ry 0 rz 180 deg; joints [-143.088, 58.823, -65.49, 142.901, 84.674, 4.016]
  MoveL 1604 to (-40.59, 150.67, 41.04) mm, rotated rx 180 ry 0 rz 180 deg; joints [-143.088, 58.823, -65.49, 142.901, 84.674, 4.016]
  Call Extruder(4.85364)
  MoveL 1605 to (-40.64, 150.37, 41.04) mm, rotated rx 180 ry 0 rz 180 deg; joints [-143.15, 58.816, -65.5, 142.963, 84.656, 4.02]
  MoveL 1606 to (-40.64, 150.37, 41.04) mm, rotated rx 180 ry 0 rz 180 deg; joints [-143.15, 58.816, -65.5, 142.963, 84.656, 4.02]
  Call Extruder(5.01464)
  MoveL 1607 to (-40.69, 150.06, 41.04) mm, rotated rx -180 ry 0 rz 180 deg; joints [-143.213, 58.808, -65.51, 143.024, 84.637, 4.025]
  MoveL 1608 to (-40.69, 150.06, 41.04) mm, rotated rx -180 ry 0 rz 180 deg; joints [-143.213, 58.808, -65.51, 143.024, 84.637, 4.025]
  Call Extruder(5.17491)
  MoveL 1609 to (-40.74, 149.76, 41.04) mm, rotated rx 180 ry 0 rz 180 deg; joints [-143.276, 58.801, -65.52, 143.086, 84.619, 4.03]
  MoveL 1610 to (-40.74, 149.76, 41.04) mm, rotated rx 180 ry 0 rz 180 deg; joints [-143.276, 58.801, -65.52, 143.086, 84.619, 4.03]
  Call Extruder(5.33445)
  MoveL 1611 to (-40.78, 149.45, 41.04) mm, rotated rx -180 ry 0 rz 180 deg; joints [-143.338, 58.793, -65.529, 143.148, 84.601, 4.034]
  MoveL 1612 to (-40.78, 149.45, 41.04) mm, rotated rx -180 ry 0 rz 180 deg; joints [-143.338, 58.793, -65.529, 143.148, 84.601, 4.034]
  Call Extruder(5.49326)
  MoveL 1613 to (-40.83, 149.14, 41.04) mm, rotated rx 180 ry 0 rz 180 deg; joints [-143.401, 58.785, -65.539, 143.21, 84.582, 4.039]
  MoveL 1614 to (-40.83, 149.14, 41.04) mm, rotated rx 180 ry 0 rz 180 deg; joints [-143.401, 58.785, -65.539, 143.21, 84.582, 4.039]
  Call Extruder(5.67193)
  MoveL 1615 to (-40.88, 148.8, 41.04) mm, rotated rx 180 ry 0 rz -180 deg; joints [-143.471, 58.776, -65.551, 143.279, 84.561, 4.044]
  MoveL 1616 to (-40.88, 148.8, 41.04) mm, rotated rx 180 ry 0 rz -180 deg; joints [-143.471, 58.776, -65.551, 143.279, 84.561, 4.044]
  Call Extruder(5.87037)
  MoveL 1617 to (-40.93, 148.41, 41.04) mm, rotated rx -180 ry 0 rz 180 deg; joints [-143.549, 58.766, -65.564, 143.356, 84.537, 4.051]
  MoveL 1618 to (-40.93, 148.41, 41.04) mm, rotated rx -180 ry 0 rz 180 deg; joints [-143.549, 58.766, -65.564, 143.356, 84.537, 4.051]
  Call Extruder(6.06794)
  MoveL 1619 to (-40.97, 148.02, 41.04) mm, rotated rx -180 ry 0 rz 180 deg; joints [-143.627, 58.756, -65.577, 143.432, 84.513, 4.057]
  MoveL 1620 to (-40.97, 148.02, 41.04) mm, rotated rx -180 ry 0 rz 180 deg; joints [-143.627, 58.756, -65.577, 143.432, 84.513, 4.057]
  Call Extruder(6.26465)
  MoveL 1621 to (-41.02, 147.63, 41.04) mm, rotated rx -180 ry 0 rz -180 deg; joints [-143.705, 58.746, -65.59, 143.509, 84.488, 4.064]
  MoveL 1622 to (-41.02, 147.63, 41.04) mm, rotated rx -180 ry 0 rz -180 deg; joints [-143.705, 58.746, -65.59, 143.509, 84.488, 4.064]
  Call Extruder(6.46049)
  MoveL 1623 to (-41.06, 147.25, 41.04) mm, rotated rx 180 ry 0 rz -180 deg; joints [-143.783, 58.735, -65.603, 143.586, 84.464, 4.07]
  MoveL 1624 to (-41.06, 147.25, 41.04) mm, rotated rx 180 ry 0 rz -180 deg; joints [-143.783, 58.735, -65.603, 143.586, 84.464, 4.07]
  Call Extruder(6.75588)
  MoveL 1625 to (-41.11, 146.66, 41.04) mm, rotated rx -180 ry 0 rz -180 deg; joints [-143.899, 58.719, -65.624, 143.7, 84.426, 4.081]
  MoveL 1626 to (-41.11, 146.66, 41.04) mm, rotated rx -180 ry 0 rz -180 deg; joints [-143.899, 58.719, -65.624, 143.7, 84.426, 4.081]
  Call Extruder(7.04995)
  MoveL 1627 to (-41.15, 146.07, 41.04) mm, rotated rx -180 ry 0 rz 180 deg; joints [-144.015, 58.702, -65.644, 143.814, 84.388, 4.092]
  MoveL 1628 to (-41.15, 146.07, 41.04) mm, rotated rx -180 ry 0 rz 180 deg; joints [-144.015, 58.702, -65.644, 143.814, 84.388, 4.092]
  Call Extruder(7.34268)
  MoveL 1629 to (-41.2, 145.48, 41.04) mm, rotated rx -180 ry 0 rz 180 deg; joints [-144.131, 58.686, -65.665, 143.929, 84.349, 4.103]
  MoveL 1630 to (-41.2, 145.48, 41.04) mm, rotated rx -180 ry 0 rz 180 deg; joints [-144.131, 58.686, -65.665, 143.929, 84.349, 4.103]
  Call Extruder(7.91614)
  MoveL 1631 to (-41.25, 144.32, 41.04) mm, rotated rx 180 ry 0 rz 180 deg; joints [-144.355, 58.651, -65.708, 144.149, 84.271, 4.126]
  MoveL 1632 to (-41.25, 144.32, 41.04) mm, rotated rx 180 ry 0 rz 180 deg; joints [-144.355, 58.651, -65.708, 144.149, 84.271, 4.126]
  Call Extruder(8.63010)
  MoveL 1633 to (-41.29, 142.86, 41.04) mm, rotated rx 180 ry 0 rz -180 deg; joints [-144.635, 58.608, -65.762, 144.424, 84.171, 4.155]
  Call Extruder(50.69492)
  MoveL 1634 to (-41.29, 57.14, 41.04) mm, rotated rx 180 ry 0 rz 180 deg; joints [-164.153, 56.367, -67.977, 163.839, 78.838, 3.211]
  Call Extruder(51.12347)
  MoveL 1635 to (-41.27, 56.26, 41.04) mm, rotated rx -180 ry 0 rz -180 deg; joints [-164.382, 56.351, -67.99, 164.071, 78.796, 3.174]
  MoveL 1636 to (-41.27, 56.26, 41.04) mm, rotated rx -180 ry 0 rz -180 deg; joints [-164.382, 56.351, -67.99, 164.071, 78.796, 3.174]
  Call Extruder(51.69692)
  MoveL 1637 to (-41.23, 55.1, 41.04) mm, rotated rx 180 ry 0 rz 180 deg; joints [-164.686, 56.328, -68.008, 164.378, 78.74, 3.125]
  MoveL 1638 to (-41.23, 55.1, 41.04) mm, rotated rx 180 ry 0 rz 180 deg; joints [-164.686, 56.328, -68.008, 164.378, 78.74, 3.125]
  Call Extruder(52.13124)
  MoveL 1639 to (-41.18, 54.23, 41.04) mm, rotated rx -180 ry 0 rz 180 deg; joints [-164.915, 56.31, -68.022, 164.609, 78.697, 3.088]
  MoveL 1640 to (-41.18, 54.23, 41.04) mm, rotated rx -180 ry 0 rz 180 deg; joints [-164.915, 56.31, -68.022, 164.609, 78.697, 3.088]
  Call Extruder(52.42530)
  MoveL 1641 to (-41.13, 53.64, 41.04) mm, rotated rx -180 ry 0 rz 180 deg; joints [-165.068, 56.297, -68.032, 164.764, 78.666, 3.064]
  MoveL 1642 to (-41.13, 53.64, 41.04) mm, rotated rx -180 ry 0 rz 180 deg; joints [-165.068, 56.297, -68.032, 164.764, 78.666, 3.064]
  Call Extruder(52.72070)
  MoveL 1643 to (-41.09, 53.05, 41.04) mm, rotated rx -180 ry 0 rz -180 deg; joints [-165.222, 56.284, -68.042, 164.919, 78.636, 3.039]
  MoveL 1644 to (-41.09, 53.05, 41.04) mm, rotated rx -180 ry 0 rz -180 deg; joints [-165.222, 56.284, -68.042, 164.919, 78.636, 3.039]
  Call Extruder(52.96694)
  MoveL 1645 to (-41.04, 52.56, 41.04) mm, rotated rx -180 ry 0 rz -180 deg; joints [-165.349, 56.273, -68.051, 165.048, 78.611, 3.019]
  MoveL 1646 to (-41.04, 52.56, 41.04) mm, rotated rx -180 ry 0 rz -180 deg; joints [-165.349, 56.273, -68.051, 165.048, 78.611, 3.019]
  Call Extruder(53.16365)
  MoveL 1647 to (-40.99, 52.17, 41.04) mm, rotated rx 180 ry 0 rz 180 deg; joints [-165.449, 56.264, -68.058, 165.149, 78.589, 3.003]
  MoveL 1648 to (-40.99, 52.17, 41.04) mm, rotated rx 180 ry 0 rz 180 deg; joints [-165.449, 56.264, -68.058, 165.149, 78.589, 3.003]
  Call Extruder(53.36122)
  MoveL 1649 to (-40.95, 51.78, 41.04) mm, rotated rx -180 ry 0 rz -180 deg; joints [-165.549, 56.254, -68.065, 165.25, 78.568, 2.987]
  MoveL 1650 to (-40.95, 51.78, 41.04) mm, rotated rx -180 ry 0 rz -180 deg; joints [-165.549, 56.254, -68.065, 165.25, 78.568, 2.987]
  Call Extruder(53.55966)
  MoveL 1651 to (-40.9, 51.4, 41.04) mm, rotated rx 180 ry 0 rz 180 deg; joints [-165.65, 56.245, -68.072, 165.352, 78.547, 2.971]
  MoveL 1652 to (-40.9, 51.4, 41.04) mm, rotated rx 180 ry 0 rz 180 deg; joints [-165.65, 56.245, -68.072, 165.352, 78.547, 2.971]
  Call Extruder(53.75897)
  MoveL 1653 to (-40.86, 51.01, 41.04) mm, rotated rx -180 ry 0 rz -180 deg; joints [-165.751, 56.236, -68.079, 165.454, 78.526, 2.955]
  MoveL 1654 to (-40.86, 51.01, 41.04) mm, rotated rx -180 ry 0 rz -180 deg; joints [-165.751, 56.236, -68.079, 165.454, 78.526, 2.955]
  Call Extruder(53.91779)
  MoveL 1655 to (-40.81, 50.7, 41.04) mm, rotated rx -180 ry 0 rz -180 deg; joints [-165.829, 56.228, -68.085, 165.533, 78.508, 2.942]
  MoveL 1656 to (-40.81, 50.7, 41.04) mm, rotated rx -180 ry 0 rz -180 deg; joints [-165.829, 56.228, -68.085, 165.533, 78.508, 2.942]
  Call Extruder(54.07733)
  MoveL 1657 to (-40.76, 50.4, 41.04) mm, rotated rx 180 ry 0 rz -180 deg; joints [-165.908, 56.22, -68.092, 165.613, 78.491, 2.93]
  MoveL 1658 to (-40.76, 50.4, 41.04) mm, rotated rx 180 ry 0 rz -180 deg; joints [-165.908, 56.22, -68.092, 165.613, 78.491, 2.93]
  Call Extruder(54.23760)
  MoveL 1659 to (-40.71, 50.09, 41.04) mm, rotated rx -180 ry 0 rz 180 deg; joints [-165.987, 56.212, -68.098, 165.692, 78.473, 2.918]
  MoveL 1660 to (-40.71, 50.09, 41.04) mm, rotated rx -180 ry 0 rz 180 deg; joints [-165.987, 56.212, -68.098, 165.692, 78.473, 2.918]
  Call Extruder(54.39860)
  MoveL 1661 to (-40.66, 49.79, 41.04) mm, rotated rx -180 ry 0 rz -180 deg; joints [-166.066, 56.204, -68.104, 165.772, 78.455, 2.905]
  MoveL 1662 to (-40.66, 49.79, 41.04) mm, rotated rx -180 ry 0 rz -180 deg; joints [-166.066, 56.204, -68.104, 165.772, 78.455, 2.905]
  Call Extruder(54.56032)
  MoveL 1663 to (-40.61, 49.48, 41.04) mm, rotated rx 180 ry 0 rz 180 deg; joints [-166.145, 56.196, -68.11, 165.852, 78.438, 2.892]
  MoveL 1664 to (-40.61, 49.48, 41.04) mm, rotated rx 180 ry 0 rz 180 deg; joints [-166.145, 56.196, -68.11, 165.852, 78.438, 2.892]
  Call Extruder(54.72278)
  MoveL 1665 to (-40.57, 49.17, 41.04) mm, rotated rx 180 ry 0 rz -180 deg; joints [-166.224, 56.188, -68.116, 165.932, 78.42, 2.88]
  MoveL 1666 to (-40.57, 49.17, 41.04) mm, rotated rx 180 ry 0 rz -180 deg; joints [-166.224, 56.188, -68.116, 165.932, 78.42, 2.88]
  Call Extruder(54.85670)
  MoveL 1667 to (-40.52, 48.92, 41.04) mm, rotated rx -180 ry 0 rz -180 deg; joints [-166.288, 56.181, -68.121, 165.997, 78.405, 2.87]
  MoveL 1668 to (-40.52, 48.92, 41.04) mm, rotated rx -180 ry 0 rz -180 deg; joints [-166.288, 56.181, -68.121, 165.997, 78.405, 2.87]
  Call Extruder(54.99124)
  MoveL 1669 to (-40.47, 48.68, 41.04) mm, rotated rx -180 ry 0 rz -180 deg; joints [-166.352, 56.174, -68.127, 166.061, 78.39, 2.86]
  MoveL 1670 to (-40.47, 48.68, 41.04) mm, rotated rx -180 ry 0 rz -180 deg; joints [-166.352, 56.174, -68.127, 166.061, 78.39, 2.86]
  Call Extruder(55.12638)
  MoveL 1671 to (-40.42, 48.43, 41.04) mm, rotated rx 180 ry 0 rz 180 deg; joints [-166.416, 56.167, -68.132, 166.126, 78.374, 2.85]
  MoveL 1672 to (-40.42, 48.43, 41.04) mm, rotated rx 180 ry 0 rz 180 deg; joints [-166.416, 56.167, -68.132, 166.126, 78.374, 2.85]
  Call Extruder(55.26214)
  MoveL 1673 to (-40.37, 48.18, 41.04) mm, rotated rx 180 ry 0 rz 180 deg; joints [-166.48, 56.16, -68.138, 166.19, 78.359, 2.839]
  MoveL 1674 to (-40.37, 48.18, 41.04) mm, rotated rx 180 ry 0 rz 180 deg; joints [-166.48, 56.16, -68.138, 166.19, 78.359, 2.839]
  Call Extruder(55.39850)
  MoveL 1675 to (-40.32, 47.93, 41.04) mm, rotated rx 180 ry 0 rz 180 deg; joints [-166.544, 56.153, -68.143, 166.255, 78.344, 2.829]
  MoveL 1676 to (-40.32, 47.93, 41.04) mm, rotated rx 180 ry 0 rz 180 deg; joints [-166.544, 56.153, -68.143, 166.255, 78.344, 2.829]
  Call Extruder(55.53548)
  MoveL 1677 to (-40.27, 47.68, 41.04) mm, rotated rx -180 ry 0 rz 180 deg; joints [-166.608, 56.146, -68.148, 166.32, 78.329, 2.819]
  MoveL 1678 to (-40.27, 47.68, 41.04) mm, rotated rx -180 ry 0 rz 180 deg; joints [-166.608, 56.146, -68.148, 166.32, 78.329, 2.819]
  Call Extruder(55.67306)
  MoveL 1679 to (-40.22, 47.43, 41.04) mm, rotated rx -180 ry 0 rz 180 deg; joints [-166.673, 56.139, -68.153, 166.385, 78.314, 2.809]
  MoveL 1680 to (-40.22, 47.43, 41.04) mm, rotated rx -180 ry 0 rz 180 deg; joints [-166.673, 56.139, -68.153, 166.385, 78.314, 2.809]
  Call Extruder(55.78679)
  MoveL 1681 to (-40.17, 47.23, 41.04) mm, rotated rx -180 ry 0 rz 180 deg; joints [-166.725, 56.133, -68.158, 166.438, 78.301, 2.8]
  MoveL 1682 to (-40.17, 47.23, 41.04) mm, rotated rx -180 ry 0 rz 180 deg; joints [-166.725, 56.133, -68.158, 166.438, 78.301, 2.8]
  Call Extruder(55.90097)
  MoveL 1683 to (-40.13, 47.02, 41.04) mm, rotated rx -180 ry 0 rz 180 deg; joints [-166.778, 56.127, -68.163, 166.491, 78.288, 2.792]
  MoveL 1684 to (-40.13, 47.02, 41.04) mm, rotated rx -180 ry 0 rz 180 deg; joints [-166.778, 56.127, -68.163, 166.491, 78.288, 2.792]
  Call Extruder(56.01561)
  MoveL 1685 to (-40.08, 46.82, 41.04) mm, rotated rx -180 ry 0 rz -180 deg; joints [-166.83, 56.121, -68.167, 166.544, 78.275, 2.784]
  MoveL 1686 to (-40.08, 46.82, 41.04) mm, rotated rx -180 ry 0 rz -180 deg; joints [-166.83, 56.121, -68.167, 166.544, 78.275, 2.784]
  Call Extruder(56.13069)
  MoveL 1687 to (-40.04, 46.61, 41.04) mm, rotated rx -180 ry 0 rz 180 deg; joints [-166.883, 56.115, -68.172, 166.598, 78.263, 2.775]
  MoveL 1688 to (-40.04, 46.61, 41.04) mm, rotated rx -180 ry 0 rz 180 deg; joints [-166.883, 56.115, -68.172, 166.598, 78.263, 2.775]
  Call Extruder(56.25293)
  MoveL 1689 to (-39.98, 46.4, 41.03) mm, rotated rx 180 ry 0 rz -180 deg; joints [-166.937, 56.108, -68.177, 166.653, 78.248, 2.767]
  MoveL 1690 to (-39.98, 46.4, 41.03) mm, rotated rx 180 ry 0 rz -180 deg; joints [-166.937, 56.108, -68.177, 166.653, 78.248, 2.767]
  Call Extruder(56.38259)
  MoveL 1691 to (-39.92, 46.18, 41.04) mm, rotated rx -180 ry 0 rz -180 deg; joints [-166.994, 56.101, -68.182, 166.71, 78.233, 2.758]
  MoveL 1692 to (-39.92, 46.18, 41.04) mm, rotated rx -180 ry 0 rz -180 deg; joints [-166.994, 56.101, -68.182, 166.71, 78.233, 2.758]
  Call Extruder(56.51282)
  MoveL 1693 to (-39.85, 45.95, 41.04) mm, rotated rx 180 ry 0 rz -180 deg; joints [-167.051, 56.093, -68.188, 166.767, 78.217, 2.749]
  MoveL 1694 to (-39.85, 45.95, 41.04) mm, rotated rx 180 ry 0 rz -180 deg; joints [-167.051, 56.093, -68.188, 166.767, 78.217, 2.749]
  Call Extruder(56.64361)
  MoveL 1695 to (-39.78, 45.73, 41.04) mm, rotated rx 180 ry 0 rz -180 deg; joints [-167.107, 56.085, -68.194, 166.824, 78.201, 2.741]
  MoveL 1696 to (-39.78, 45.73, 41.04) mm, rotated rx 180 ry 0 rz -180 deg; joints [-167.107, 56.085, -68.194, 166.824, 78.201, 2.741]
  Call Extruder(56.77497)
  MoveL 1697 to (-39.71, 45.5, 41.04) mm, rotated rx -180 ry 0 rz 180 deg; joints [-167.164, 56.078, -68.2, 166.881, 78.185, 2.732]
  MoveL 1698 to (-39.71, 45.5, 41.04) mm, rotated rx -180 ry 0 rz 180 deg; joints [-167.164, 56.078, -68.2, 166.881, 78.185, 2.732]
  Call Extruder(56.88687)
  MoveL 1699 to (-39.65, 45.32, 41.04) mm, rotated rx 180 ry 0 rz 180 deg; joints [-167.212, 56.071, -68.205, 166.929, 78.171, 2.725]
  MoveL 1700 to (-39.65, 45.32, 41.04) mm, rotated rx 180 ry 0 rz 180 deg; joints [-167.212, 56.071, -68.205, 166.929, 78.171, 2.725]
  Call Extruder(56.99922)
  MoveL 1701 to (-39.59, 45.13, 41.03) mm, rotated rx -180 ry 0 rz -180 deg; joints [-167.26, 56.064, -68.21, 166.978, 78.158, 2.717]
  MoveL 1702 to (-39.59, 45.13, 41.03) mm, rotated rx -180 ry 0 rz -180 deg; joints [-167.26, 56.064, -68.21, 166.978, 78.158, 2.717]
  Call Extruder(57.11201)
  MoveL 1703 to (-39.53, 44.94, 41.04) mm, rotated rx 180 ry 0 rz 180 deg; joints [-167.307, 56.057, -68.215, 167.026, 78.144, 2.71]
  MoveL 1704 to (-39.53, 44.94, 41.04) mm, rotated rx 180 ry 0 rz 180 deg; joints [-167.307, 56.057, -68.215, 167.026, 78.144, 2.71]
  Call Extruder(57.22525)
  MoveL 1705 to (-39.47, 44.75, 41.04) mm, rotated rx -180 ry 0 rz 180 deg; joints [-167.355, 56.051, -68.22, 167.074, 78.13, 2.703]
  MoveL 1706 to (-39.47, 44.75, 41.04) mm, rotated rx -180 ry 0 rz 180 deg; joints [-167.355, 56.051, -68.22, 167.074, 78.13, 2.703]
  Call Extruder(57.33893)
  MoveL 1707 to (-39.41, 44.56, 41.04) mm, rotated rx 180 ry 0 rz -180 deg; joints [-167.403, 56.044, -68.225, 167.122, 78.117, 2.695]
  MoveL 1708 to (-39.41, 44.56, 41.04) mm, rotated rx 180 ry 0 rz -180 deg; joints [-167.403, 56.044, -68.225, 167.122, 78.117, 2.695]
  Call Extruder(57.52088)
  MoveL 1709 to (-39.29, 44.27, 41.04) mm, rotated rx 180 ry 0 rz 180 deg; joints [-167.475, 56.032, -68.234, 167.195, 78.093, 2.685]
  MoveL 1710 to (-39.29, 44.27, 41.04) mm, rotated rx 180 ry 0 rz 180 deg; joints [-167.475, 56.032, -68.234, 167.195, 78.093, 2.685]
  Call Extruder(57.70360)
  MoveL 1711 to (-39.17, 43.98, 41.04) mm, rotated rx -180 ry 0 rz 180 deg; joints [-167.548, 56.02, -68.243, 167.268, 78.069, 2.674]
  MoveL 1712 to (-39.17, 43.98, 41.04) mm, rotated rx -180 ry 0 rz 180 deg; joints [-167.548, 56.02, -68.243, 167.268, 78.069, 2.674]
  Call Extruder(57.87401)
  MoveL 1713 to (-39.05, 43.71, 41.04) mm, rotated rx -180 ry 0 rz -180 deg; joints [-167.615, 56.008, -68.251, 167.336, 78.046, 2.665]
  MoveL 1714 to (-39.05, 43.71, 41.04) mm, rotated rx -180 ry 0 rz -180 deg; joints [-167.615, 56.008, -68.251, 167.336, 78.046, 2.665]
  Call Extruder(58.03200)
  MoveL 1715 to (-38.94, 43.46, 41.04) mm, rotated rx -180 ry 0 rz -180 deg; joints [-167.677, 55.998, -68.259, 167.399, 78.026, 2.656]
  MoveL 1716 to (-38.94, 43.46, 41.04) mm, rotated rx -180 ry 0 rz -180 deg; joints [-167.677, 55.998, -68.259, 167.399, 78.026, 2.656]
  Call Extruder(58.19059)
  MoveL 1717 to (-38.84, 43.21, 41.04) mm, rotated rx -180 ry 0 rz -180 deg; joints [-167.739, 55.987, -68.267, 167.461, 78.005, 2.646]
  MoveL 1718 to (-38.84, 43.21, 41.04) mm, rotated rx -180 ry 0 rz -180 deg; joints [-167.739, 55.987, -68.267, 167.461, 78.005, 2.646]
  Call Extruder(58.39676)
  MoveL 1719 to (-38.66, 42.91, 41.04) mm, rotated rx -180 ry 0 rz -180 deg; joints [-167.813, 55.972, -68.278, 167.535, 77.975, 2.637]
  MoveL 1720 to (-38.66, 42.91, 41.04) mm, rotated rx -180 ry 0 rz -180 deg; joints [-167.813, 55.972, -68.278, 167.535, 77.975, 2.637]
  Call Extruder(58.60370)
  MoveL 1721 to (-38.49, 42.6, 41.04) mm, rotated rx -180 ry 0 rz 180 deg; joints [-167.886, 55.956, -68.29, 167.609, 77.945, 2.627]
  MoveL 1722 to (-38.49, 42.6, 41.04) mm, rotated rx -180 ry 0 rz 180 deg; joints [-167.886, 55.956, -68.29, 167.609, 77.945, 2.627]
  Call Extruder(58.81142)
  MoveL 1723 to (-38.31, 42.3, 41.04) mm, rotated rx -180 ry 0 rz 180 deg; joints [-167.96, 55.94, -68.302, 167.683, 77.915, 2.617]
  MoveL 1724 to (-38.31, 42.3, 41.04) mm, rotated rx -180 ry 0 rz 180 deg; joints [-167.96, 55.94, -68.302, 167.683, 77.915, 2.617]
  Call Extruder(59.01993)
  MoveL 1725 to (-38.13, 41.99, 41.04) mm, rotated rx -180 ry 0 rz -180 deg; joints [-168.033, 55.924, -68.313, 167.757, 77.885, 2.608]
  MoveL 1726 to (-38.13, 41.99, 41.04) mm, rotated rx -180 ry 0 rz -180 deg; joints [-168.033, 55.924, -68.313, 167.757, 77.885, 2.608]
  Call Extruder(59.19948)
  MoveL 1727 to (-37.96, 41.75, 41.04) mm, rotated rx -180 ry 0 rz -180 deg; joints [-168.091, 55.91, -68.324, 167.814, 77.857, 2.601]
  MoveL 1728 to (-37.96, 41.75, 41.04) mm, rotated rx -180 ry 0 rz -180 deg; joints [-168.091, 55.91, -68.324, 167.814, 77.857, 2.601]
  Call Extruder(59.53291)
  MoveL 1729 to (-37.63, 41.3, 41.04) mm, rotated rx -180 ry 0 rz -180 deg; joints [-168.197, 55.882, -68.344, 167.92, 77.805, 2.588]
  MoveL 1730 to (-37.63, 41.3, 41.04) mm, rotated rx -180 ry 0 rz -180 deg; joints [-168.197, 55.882, -68.344, 167.92, 77.805, 2.588]
  Call Extruder(59.86753)
  MoveL 1731 to (-37.3, 40.85, 41.04) mm, rotated rx -180 ry 0 rz -180 deg; joints [-168.304, 55.854, -68.364, 168.027, 77.754, 2.575]
  Call Extruder(60.69546)
  MoveL 1732 to (-36.39, 39.81, 41.04) mm, rotated rx -180 ry 0 rz 180 deg; joints [-168.541, 55.78, -68.417, 168.265, 77.618, 2.55]
  Call Extruder(61.52337)
  MoveL 1733 to (-35.35, 38.9, 41.04) mm, rotated rx 180 ry 0 rz 180 deg; joints [-168.739, 55.699, -68.474, 168.461, 77.474, 2.535]
  Call Extruder(61.69068)
  MoveL 1734 to (-35.13, 38.73, 41.04) mm, rotated rx 180 ry 0 rz 180 deg; joints [-168.773, 55.681, -68.487, 168.494, 77.444, 2.534]
  MoveL 1735 to (-35.13, 38.73, 41.04) mm, rotated rx 180 ry 0 rz 180 deg; joints [-168.773, 55.681, -68.487, 168.494, 77.444, 2.534]
  Call Extruder(62.02410)
  MoveL 1736 to (-34.68, 38.4, 41.04) mm, rotated rx -180 ry 0 rz 180 deg; joints [-168.84, 55.647, -68.511, 168.56, 77.384, 2.531]
  MoveL 1737 to (-34.68, 38.4, 41.04) mm, rotated rx -180 ry 0 rz 180 deg; joints [-168.84, 55.647, -68.511, 168.56, 77.384, 2.531]
  Call Extruder(62.35635)
  MoveL 1738 to (-34.23, 38.08, 41.04) mm, rotated rx 180 ry 0 rz -180 deg; joints [-168.908, 55.612, -68.534, 168.628, 77.323, 2.527]
  MoveL 1739 to (-34.23, 38.08, 41.04) mm, rotated rx 180 ry 0 rz -180 deg; joints [-168.908, 55.612, -68.534, 168.628, 77.323, 2.527]
  Call Extruder(62.47405)
  MoveL 1740 to (-34.05, 37.98, 41.04) mm, rotated rx -180 ry 0 rz 180 deg; joints [-168.927, 55.6, -68.543, 168.646, 77.301, 2.527]
  MoveL 1741 to (-34.05, 37.98, 41.04) mm, rotated rx -180 ry 0 rz 180 deg; joints [-168.927, 55.6, -68.543, 168.646, 77.301, 2.527]
  Call Extruder(62.68177)
  MoveL 1742 to (-33.75, 37.8, 41.04) mm, rotated rx -180 ry 0 rz -180 deg; joints [-168.96, 55.577, -68.559, 168.678, 77.262, 2.528]
  MoveL 1743 to (-33.75, 37.8, 41.04) mm, rotated rx -180 ry 0 rz -180 deg; joints [-168.96, 55.577, -68.559, 168.678, 77.262, 2.528]
  Call Extruder(62.88871)
  MoveL 1744 to (-33.45, 37.63, 41.04) mm, rotated rx -180 ry 0 rz 180 deg; joints [-168.993, 55.554, -68.574, 168.71, 77.223, 2.528]
  MoveL 1745 to (-33.45, 37.63, 41.04) mm, rotated rx -180 ry 0 rz 180 deg; joints [-168.993, 55.554, -68.574, 168.71, 77.223, 2.528]
  Call Extruder(63.09487)
  MoveL 1746 to (-33.14, 37.45, 41.03) mm, rotated rx 180 ry 0 rz 180 deg; joints [-169.026, 55.531, -68.59, 168.742, 77.184, 2.528]
  MoveL 1747 to (-33.14, 37.45, 41.03) mm, rotated rx 180 ry 0 rz 180 deg; joints [-169.026, 55.531, -68.59, 168.742, 77.184, 2.528]
  Call Extruder(63.27655)
  MoveL 1748 to (-32.87, 37.31, 41.04) mm, rotated rx -180 ry 0 rz -180 deg; joints [-169.052, 55.511, -68.604, 168.767, 77.15, 2.529]
  MoveL 1749 to (-32.87, 37.31, 41.04) mm, rotated rx -180 ry 0 rz -180 deg; joints [-169.052, 55.511, -68.604, 168.767, 77.15, 2.529]
  Call Extruder(63.43455)
  MoveL 1750 to (-32.62, 37.2, 41.04) mm, rotated rx 180 ry 0 rz 180 deg; joints [-169.068, 55.493, -68.616, 168.783, 77.119, 2.531]
  MoveL 1751 to (-32.62, 37.2, 41.04) mm, rotated rx 180 ry 0 rz 180 deg; joints [-169.068, 55.493, -68.616, 168.783, 77.119, 2.531]
  Call Extruder(63.59195)
  MoveL 1752 to (-32.37, 37.09, 41.04) mm, rotated rx 180 ry 0 rz 180 deg; joints [-169.085, 55.474, -68.628, 168.799, 77.088, 2.534]
  MoveL 1753 to (-32.37, 37.09, 41.04) mm, rotated rx 180 ry 0 rz 180 deg; joints [-169.085, 55.474, -68.628, 168.799, 77.088, 2.534]
  Call Extruder(63.77466)
  MoveL 1754 to (-32.08, 36.97, 41.04) mm, rotated rx -180 ry 0 rz 180 deg; joints [-169.104, 55.453, -68.643, 168.816, 77.052, 2.537]
  MoveL 1755 to (-32.08, 36.97, 41.04) mm, rotated rx -180 ry 0 rz 180 deg; joints [-169.104, 55.453, -68.643, 168.816, 77.052, 2.537]
  Call Extruder(63.95661)
  MoveL 1756 to (-31.78, 36.85, 41.04) mm, rotated rx -180 ry 0 rz 180 deg; joints [-169.122, 55.432, -68.657, 168.833, 77.017, 2.539]
  MoveL 1757 to (-31.78, 36.85, 41.04) mm, rotated rx -180 ry 0 rz 180 deg; joints [-169.122, 55.432, -68.657, 168.833, 77.017, 2.539]
  Call Extruder(64.10394)
  MoveL 1758 to (-31.54, 36.76, 41.03) mm, rotated rx -180 ry 0 rz 180 deg; joints [-169.135, 55.414, -68.669, 168.845, 76.988, 2.542]
  MoveL 1759 to (-31.54, 36.76, 41.03) mm, rotated rx -180 ry 0 rz 180 deg; joints [-169.135, 55.414, -68.669, 168.845, 76.988, 2.542]
  Call Extruder(64.21718)
  MoveL 1760 to (-31.35, 36.7, 41.04) mm, rotated rx 180 ry 0 rz 180 deg; joints [-169.143, 55.401, -68.678, 168.852, 76.965, 2.545]
  MoveL 1761 to (-31.35, 36.7, 41.04) mm, rotated rx 180 ry 0 rz 180 deg; joints [-169.143, 55.401, -68.678, 168.852, 76.965, 2.545]
  Call Extruder(64.32997)
  MoveL 1762 to (-31.17, 36.64, 41.04) mm, rotated rx -180 ry 0 rz 180 deg; joints [-169.15, 55.387, -68.687, 168.858, 76.943, 2.548]
  MoveL 1763 to (-31.17, 36.64, 41.04) mm, rotated rx -180 ry 0 rz 180 deg; joints [-169.15, 55.387, -68.687, 168.858, 76.943, 2.548]
  Call Extruder(64.44232)
  MoveL 1764 to (-30.98, 36.58, 41.03) mm, rotated rx -180 ry 0 rz 180 deg; joints [-169.157, 55.374, -68.696, 168.865, 76.92, 2.551]
  MoveL 1765 to (-30.98, 36.58, 41.03) mm, rotated rx -180 ry 0 rz 180 deg; joints [-169.157, 55.374, -68.696, 168.865, 76.92, 2.551]
  Call Extruder(64.55422)
  MoveL 1766 to (-30.79, 36.52, 41.04) mm, rotated rx -180 ry 0 rz 180 deg; joints [-169.164, 55.36, -68.705, 168.871, 76.898, 2.553]
  MoveL 1767 to (-30.79, 36.52, 41.04) mm, rotated rx -180 ry 0 rz 180 deg; joints [-169.164, 55.36, -68.705, 168.871, 76.898, 2.553]
  Call Extruder(64.67562)
  MoveL 1768 to (-30.58, 36.45, 41.04) mm, rotated rx 180 ry 0 rz 180 deg; joints [-169.172, 55.345, -68.714, 168.878, 76.873, 2.557]
  MoveL 1769 to (-30.58, 36.45, 41.04) mm, rotated rx 180 ry 0 rz 180 deg; joints [-169.172, 55.345, -68.714, 168.878, 76.873, 2.557]
  Call Extruder(64.80641)
  MoveL 1770 to (-30.36, 36.38, 41.04) mm, rotated rx -180 ry 0 rz 180 deg; joints [-169.179, 55.329, -68.725, 168.884, 76.846, 2.56]
  MoveL 1771 to (-30.36, 36.38, 41.04) mm, rotated rx -180 ry 0 rz 180 deg; joints [-169.179, 55.329, -68.725, 168.884, 76.846, 2.56]
  Call Extruder(64.93664)
  MoveL 1772 to (-30.14, 36.32, 41.04) mm, rotated rx -180 ry 0 rz 180 deg; joints [-169.186, 55.313, -68.735, 168.89, 76.82, 2.564]
  MoveL 1773 to (-30.14, 36.32, 41.04) mm, rotated rx -180 ry 0 rz 180 deg; joints [-169.186, 55.313, -68.735, 168.89, 76.82, 2.564]
  Call Extruder(65.06630)
  MoveL 1774 to (-29.91, 36.25, 41.04) mm, rotated rx -180 ry 0 rz -180 deg; joints [-169.193, 55.297, -68.746, 168.896, 76.793, 2.567]
  MoveL 1775 to (-29.91, 36.25, 41.04) mm, rotated rx -180 ry 0 rz -180 deg; joints [-169.193, 55.297, -68.746, 168.896, 76.793, 2.567]
  Call Extruder(65.19540)
  MoveL 1776 to (-29.69, 36.18, 41.04) mm, rotated rx 180 ry 0 rz -180 deg; joints [-169.201, 55.28, -68.757, 168.902, 76.767, 2.571]
  MoveL 1777 to (-29.69, 36.18, 41.04) mm, rotated rx 180 ry 0 rz -180 deg; joints [-169.201, 55.28, -68.757, 168.902, 76.767, 2.571]
  Call Extruder(65.31047)
  MoveL 1778 to (-29.48, 36.14, 41.04) mm, rotated rx -180 ry 0 rz 180 deg; joints [-169.202, 55.266, -68.766, 168.903, 76.743, 2.575]
  MoveL 1779 to (-29.48, 36.14, 41.04) mm, rotated rx -180 ry 0 rz 180 deg; joints [-169.202, 55.266, -68.766, 168.903, 76.743, 2.575]
  Call Extruder(65.42509)
  MoveL 1780 to (-29.28, 36.09, 41.04) mm, rotated rx -180 ry 0 rz -180 deg; joints [-169.204, 55.251, -68.775, 168.904, 76.72, 2.58]
  MoveL 1781 to (-29.28, 36.09, 41.04) mm, rotated rx -180 ry 0 rz -180 deg; joints [-169.204, 55.251, -68.775, 168.904, 76.72, 2.58]
  Call Extruder(65.53926)
  MoveL 1782 to (-29.08, 36.05, 41.04) mm, rotated rx -180 ry 0 rz 180 deg; joints [-169.206, 55.237, -68.785, 168.904, 76.696, 2.584]
  MoveL 1783 to (-29.08, 36.05, 41.04) mm, rotated rx -180 ry 0 rz 180 deg; joints [-169.206, 55.237, -68.785, 168.904, 76.696, 2.584]
  Call Extruder(65.65298)
  MoveL 1784 to (-28.87, 36, 41.04) mm, rotated rx 180 ry 0 rz 180 deg; joints [-169.207, 55.222, -68.794, 168.905, 76.672, 2.588]
  MoveL 1785 to (-28.87, 36, 41.04) mm, rotated rx 180 ry 0 rz 180 deg; joints [-169.207, 55.222, -68.794, 168.905, 76.672, 2.588]
  Call Extruder(65.77840)
  MoveL 1786 to (-28.64, 35.96, 41.04) mm, rotated rx 180 ry 0 rz -180 deg; joints [-169.208, 55.206, -68.805, 168.905, 76.646, 2.593]
  MoveL 1787 to (-28.64, 35.96, 41.04) mm, rotated rx 180 ry 0 rz -180 deg; joints [-169.208, 55.206, -68.805, 168.905, 76.646, 2.593]
  Call Extruder(65.91538)
  MoveL 1788 to (-28.4, 35.91, 41.04) mm, rotated rx -180 ry 0 rz 180 deg; joints [-169.209, 55.188, -68.816, 168.904, 76.618, 2.599]
  MoveL 1789 to (-28.4, 35.91, 41.04) mm, rotated rx -180 ry 0 rz 180 deg; joints [-169.209, 55.188, -68.816, 168.904, 76.618, 2.599]
  Call Extruder(66.05174)
  MoveL 1790 to (-28.15, 35.86, 41.04) mm, rotated rx -180 ry 0 rz -180 deg; joints [-169.21, 55.17, -68.827, 168.903, 76.589, 2.605]
  MoveL 1791 to (-28.15, 35.86, 41.04) mm, rotated rx -180 ry 0 rz -180 deg; joints [-169.21, 55.17, -68.827, 168.903, 76.589, 2.605]
  Call Extruder(66.18750)
  MoveL 1792 to (-27.9, 35.81, 41.04) mm, rotated rx -180 ry 0 rz -180 deg; joints [-169.21, 55.153, -68.839, 168.903, 76.56, 2.61]
  MoveL 1793 to (-27.9, 35.81, 41.04) mm, rotated rx -180 ry 0 rz -180 deg; joints [-169.21, 55.153, -68.839, 168.903, 76.56, 2.61]
  Call Extruder(66.32265)
  MoveL 1794 to (-27.65, 35.76, 41.04) mm, rotated rx -180 ry 0 rz -180 deg; joints [-169.211, 55.135, -68.85, 168.902, 76.532, 2.616]
  MoveL 1795 to (-27.65, 35.76, 41.04) mm, rotated rx -180 ry 0 rz -180 deg; joints [-169.211, 55.135, -68.85, 168.902, 76.532, 2.616]
  Call Extruder(66.45718)
  MoveL 1796 to (-27.4, 35.71, 41.04) mm, rotated rx 180 ry 0 rz -180 deg; joints [-169.212, 55.117, -68.861, 168.901, 76.503, 2.621]
  MoveL 1797 to (-27.4, 35.71, 41.04) mm, rotated rx 180 ry 0 rz -180 deg; joints [-169.212, 55.117, -68.861, 168.901, 76.503, 2.621]
  Call Extruder(66.59111)
  MoveL 1798 to (-27.15, 35.66, 41.04) mm, rotated rx -180 ry 0 rz 180 deg; joints [-169.212, 55.099, -68.872, 168.9, 76.475, 2.627]
  MoveL 1799 to (-27.15, 35.66, 41.04) mm, rotated rx -180 ry 0 rz 180 deg; joints [-169.212, 55.099, -68.872, 168.9, 76.475, 2.627]
  Call Extruder(66.73897)
  MoveL 1800 to (-26.87, 35.61, 41.04) mm, rotated rx 180 ry 0 rz 180 deg; joints [-169.211, 55.079, -68.885, 168.898, 76.443, 2.634]
  MoveL 1801 to (-26.87, 35.61, 41.04) mm, rotated rx 180 ry 0 rz 180 deg; joints [-169.211, 55.079, -68.885, 168.898, 76.443, 2.634]
  Call Extruder(66.90071)
  MoveL 1802 to (-26.57, 35.56, 41.04) mm, rotated rx -180 ry 0 rz 180 deg; joints [-169.208, 55.057, -68.898, 168.893, 76.409, 2.641]
  MoveL 1803 to (-26.57, 35.56, 41.04) mm, rotated rx -180 ry 0 rz 180 deg; joints [-169.208, 55.057, -68.898, 168.893, 76.409, 2.641]
  Call Extruder(67.06171)
  MoveL 1804 to (-26.26, 35.51, 41.04) mm, rotated rx -180 ry 0 rz -180 deg; joints [-169.205, 55.036, -68.912, 168.889, 76.374, 2.649]
  MoveL 1805 to (-26.26, 35.51, 41.04) mm, rotated rx -180 ry 0 rz -180 deg; joints [-169.205, 55.036, -68.912, 168.889, 76.374, 2.649]
  Call Extruder(67.22199)
  MoveL 1806 to (-25.96, 35.46, 41.04) mm, rotated rx -180 ry 0 rz 180 deg; joints [-169.202, 55.014, -68.926, 168.884, 76.339, 2.657]
  MoveL 1807 to (-25.96, 35.46, 41.04) mm, rotated rx -180 ry 0 rz 180 deg; joints [-169.202, 55.014, -68.926, 168.884, 76.339, 2.657]
  Call Extruder(67.38154)
  MoveL 1808 to (-25.65, 35.42, 41.04) mm, rotated rx 180 ry 0 rz 180 deg; joints [-169.199, 54.992, -68.939, 168.879, 76.305, 2.665]
  MoveL 1809 to (-25.65, 35.42, 41.04) mm, rotated rx 180 ry 0 rz 180 deg; joints [-169.199, 54.992, -68.939, 168.879, 76.305, 2.665]
  Call Extruder(67.54036)
  MoveL 1810 to (-25.34, 35.37, 41.04) mm, rotated rx 180 ry 0 rz 180 deg; joints [-169.196, 54.97, -68.953, 168.875, 76.27, 2.672]
  MoveL 1811 to (-25.34, 35.37, 41.04) mm, rotated rx 180 ry 0 rz 180 deg; joints [-169.196, 54.97, -68.953, 168.875, 76.27, 2.672]
  Call Extruder(67.71903)
  MoveL 1812 to (-25, 35.32, 41.04) mm, rotated rx -180 ry 0 rz -180 deg; joints [-169.191, 54.945, -68.968, 168.867, 76.231, 2.682]
  MoveL 1813 to (-25, 35.32, 41.04) mm, rotated rx -180 ry 0 rz -180 deg; joints [-169.191, 54.945, -68.968, 168.867, 76.231, 2.682]
  Call Extruder(67.91748)
  MoveL 1814 to (-24.61, 35.28, 41.03) mm, rotated rx 180 ry 0 rz 180 deg; joints [-169.182, 54.918, -68.985, 168.856, 76.188, 2.693]
  MoveL 1815 to (-24.61, 35.28, 41.03) mm, rotated rx 180 ry 0 rz 180 deg; joints [-169.182, 54.918, -68.985, 168.856, 76.188, 2.693]
  Call Extruder(68.11505)
  MoveL 1816 to (-24.22, 35.23, 41.04) mm, rotated rx -180 ry 0 rz 180 deg; joints [-169.174, 54.89, -69.001, 168.845, 76.145, 2.703]
  MoveL 1817 to (-24.22, 35.23, 41.04) mm, rotated rx -180 ry 0 rz 180 deg; joints [-169.174, 54.89, -69.001, 168.845, 76.145, 2.703]
  Call Extruder(68.31176)
  MoveL 1818 to (-23.84, 35.18, 41.04) mm, rotated rx -180 ry 0 rz 180 deg; joints [-169.166, 54.862, -69.018, 168.835, 76.102, 2.714]
  MoveL 1819 to (-23.84, 35.18, 41.04) mm, rotated rx -180 ry 0 rz 180 deg; joints [-169.166, 54.862, -69.018, 168.835, 76.102, 2.714]
  Call Extruder(68.50760)
  MoveL 1820 to (-23.45, 35.14, 41.04) mm, rotated rx -180 ry 0 rz -180 deg; joints [-169.157, 54.834, -69.035, 168.823, 76.058, 2.725]
  MoveL 1821 to (-23.45, 35.14, 41.04) mm, rotated rx -180 ry 0 rz -180 deg; joints [-169.157, 54.834, -69.035, 168.823, 76.058, 2.725]
  Call Extruder(68.80299)
  MoveL 1822 to (-22.86, 35.09, 41.04) mm, rotated rx -180 ry 0 rz 180 deg; joints [-169.137, 54.792, -69.06, 168.8, 75.994, 2.744]
  MoveL 1823 to (-22.86, 35.09, 41.04) mm, rotated rx -180 ry 0 rz 180 deg; joints [-169.137, 54.792, -69.06, 168.8, 75.994, 2.744]
  Call Extruder(69.09705)
  MoveL 1824 to (-22.27, 35.04, 41.04) mm, rotated rx -180 ry 0 rz 180 deg; joints [-169.117, 54.75, -69.085, 168.776, 75.929, 2.762]
  MoveL 1825 to (-22.27, 35.04, 41.04) mm, rotated rx -180 ry 0 rz 180 deg; joints [-169.117, 54.75, -69.085, 168.776, 75.929, 2.762]
  Call Extruder(69.38978)
  MoveL 1826 to (-21.68, 35, 41.04) mm, rotated rx -180 ry 0 rz 180 deg; joints [-169.096, 54.708, -69.11, 168.751, 75.864, 2.781]
  MoveL 1827 to (-21.68, 35, 41.04) mm, rotated rx -180 ry 0 rz 180 deg; joints [-169.096, 54.708, -69.11, 168.751, 75.864, 2.781]
  Call Extruder(69.96323)
  MoveL 1828 to (-20.52, 34.95, 41.04) mm, rotated rx -180 ry 0 rz 180 deg; joints [-169.042, 54.625, -69.158, 168.689, 75.738, 2.821]
  MoveL 1829 to (-20.52, 34.95, 41.04) mm, rotated rx -180 ry 0 rz 180 deg; joints [-169.042, 54.625, -69.158, 168.689, 75.738, 2.821]
  Call Extruder(70.67720)
  MoveL 1830 to (-19.06, 34.91, 41.04) mm, rotated rx -180 ry 0 rz -180 deg; joints [-168.967, 54.521, -69.217, 168.604, 75.582, 2.873]
  Call Extruder(187.52394)
  MoveL 1831 to (219.06, 34.91, 41.04) mm, rotated rx -180 ry 0 rz 180 deg; joints [-30.588, 44.631, -71.41, 33.509, 112.821, 14.403]
  Call Extruder(187.95250)
  MoveL 1832 to (219.94, 34.93, 41.04) mm, rotated rx 180 ry 0 rz -180 deg; joints [-30.233, 44.708, -71.412, 33.119, 112.846, 14.214]
  MoveL 1833 to (219.94, 34.93, 41.04) mm, rotated rx 180 ry 0 rz -180 deg; joints [-30.233, 44.708, -71.412, 33.119, 112.846, 14.214]
  Call Extruder(188.52594)
  MoveL 1834 to (221.1, 34.98, 41.04) mm, rotated rx -180 ry 0 rz -180 deg; joints [-29.789, 44.81, -71.414, 32.628, 112.87, 13.973]
  MoveL 1835 to (221.1, 34.98, 41.04) mm, rotated rx -180 ry 0 rz -180 deg; joints [-29.789, 44.81, -71.414, 32.628, 112.87, 13.973]
  Call Extruder(188.96026)
  MoveL 1836 to (221.97, 35.02, 41.04) mm, rotated rx -180 ry 0 rz 180 deg; joints [-29.47, 44.888, -71.415, 32.276, 112.882, 13.798]
  MoveL 1837 to (221.97, 35.02, 41.04) mm, rotated rx -180 ry 0 rz 180 deg; joints [-29.47, 44.888, -71.415, 32.276, 112.882, 13.798]
  Call Extruder(189.25431)
  MoveL 1838 to (222.56, 35.07, 41.04) mm, rotated rx -180 ry 0 rz 180 deg; joints [-29.272, 44.942, -71.416, 32.054, 112.884, 13.686]
  MoveL 1839 to (222.56, 35.07, 41.04) mm, rotated rx -180 ry 0 rz 180 deg; joints [-29.272, 44.942, -71.416, 32.054, 112.884, 13.686]
  Call Extruder(189.54970)
  MoveL 1840 to (223.15, 35.11, 41.03) mm, rotated rx -180 ry 0 rz 180 deg; joints [-29.075, 44.995, -71.416, 31.835, 112.886, 13.575]
  MoveL 1841 to (223.15, 35.11, 41.03) mm, rotated rx -180 ry 0 rz 180 deg; joints [-29.075, 44.995, -71.416, 31.835, 112.886, 13.575]
  Call Extruder(189.79594)
  MoveL 1842 to (223.64, 35.16, 41.04) mm, rotated rx 180 ry 0 rz 180 deg; joints [-28.92, 45.039, -71.417, 31.661, 112.885, 13.486]
  MoveL 1843 to (223.64, 35.16, 41.04) mm, rotated rx 180 ry 0 rz 180 deg; joints [-28.92, 45.039, -71.417, 31.661, 112.885, 13.486]
  Call Extruder(189.99264)
  MoveL 1844 to (224.03, 35.21, 41.04) mm, rotated rx -180 ry 0 rz 180 deg; joints [-28.804, 45.075, -71.417, 31.531, 112.881, 13.418]
  MoveL 1845 to (224.03, 35.21, 41.04) mm, rotated rx -180 ry 0 rz 180 deg; joints [-28.804, 45.075, -71.417, 31.531, 112.881, 13.418]
  Call Extruder(190.19022)
  MoveL 1846 to (224.42, 35.25, 41.04) mm, rotated rx -180 ry 0 rz -180 deg; joints [-28.69, 45.111, -71.417, 31.403, 112.877, 13.351]
  MoveL 1847 to (224.42, 35.25, 41.04) mm, rotated rx -180 ry 0 rz -180 deg; joints [-28.69, 45.111, -71.417, 31.403, 112.877, 13.351]
  Call Extruder(190.38866)
  MoveL 1848 to (224.8, 35.3, 41.04) mm, rotated rx -180 ry 0 rz 180 deg; joints [-28.577, 45.147, -71.418, 31.276, 112.873, 13.284]
  MoveL 1849 to (224.8, 35.3, 41.04) mm, rotated rx -180 ry 0 rz 180 deg; joints [-28.577, 45.147, -71.418, 31.276, 112.873, 13.284]
  Call Extruder(190.58797)
  MoveL 1850 to (225.19, 35.34, 41.04) mm, rotated rx 180 ry 0 rz 180 deg; joints [-28.465, 45.183, -71.418, 31.15, 112.868, 13.218]
  MoveL 1851 to (225.19, 35.34, 41.04) mm, rotated rx 180 ry 0 rz 180 deg; joints [-28.465, 45.183, -71.418, 31.15, 112.868, 13.218]
  Call Extruder(190.74679)
  MoveL 1852 to (225.5, 35.39, 41.03) mm, rotated rx -180 ry 0 rz 180 deg; joints [-28.385, 45.212, -71.418, 31.059, 112.862, 13.17]
  MoveL 1853 to (225.5, 35.39, 41.03) mm, rotated rx -180 ry 0 rz 180 deg; joints [-28.385, 45.212, -71.418, 31.059, 112.862, 13.17]
  Call Extruder(190.90634)
  MoveL 1854 to (225.8, 35.44, 41.03) mm, rotated rx 180 ry 0 rz 180 deg; joints [-28.307, 45.241, -71.418, 30.97, 112.855, 13.121]
  MoveL 1855 to (225.8, 35.44, 41.03) mm, rotated rx 180 ry 0 rz 180 deg; joints [-28.307, 45.241, -71.418, 30.97, 112.855, 13.121]
  Call Extruder(191.06662)
  MoveL 1856 to (226.11, 35.49, 41.04) mm, rotated rx -180 ry 0 rz 180 deg; joints [-28.228, 45.269, -71.418, 30.881, 112.848, 13.073]
  MoveL 1857 to (226.11, 35.49, 41.04) mm, rotated rx -180 ry 0 rz 180 deg; joints [-28.228, 45.269, -71.418, 30.881, 112.848, 13.073]
  Call Extruder(191.22762)
  MoveL 1858 to (226.41, 35.54, 41.03) mm, rotated rx 180 ry 0 rz 180 deg; joints [-28.151, 45.298, -71.418, 30.793, 112.841, 13.025]
  MoveL 1859 to (226.41, 35.54, 41.03) mm, rotated rx 180 ry 0 rz 180 deg; joints [-28.151, 45.298, -71.418, 30.793, 112.841, 13.025]
  Call Extruder(191.38936)
  MoveL 1860 to (226.72, 35.59, 41.04) mm, rotated rx -180 ry 0 rz 180 deg; joints [-28.074, 45.327, -71.418, 30.705, 112.833, 12.978]
  MoveL 1861 to (226.72, 35.59, 41.04) mm, rotated rx -180 ry 0 rz 180 deg; joints [-28.074, 45.327, -71.418, 30.705, 112.833, 12.978]
  Call Extruder(191.55182)
  MoveL 1862 to (227.03, 35.64, 41.04) mm, rotated rx -180 ry 0 rz 180 deg; joints [-27.998, 45.356, -71.418, 30.619, 112.825, 12.931]
  MoveL 1863 to (227.03, 35.64, 41.04) mm, rotated rx -180 ry 0 rz 180 deg; joints [-27.998, 45.356, -71.418, 30.619, 112.825, 12.931]
  Call Extruder(191.68574)
  MoveL 1864 to (227.28, 35.68, 41.04) mm, rotated rx -180 ry 0 rz 180 deg; joints [-27.942, 45.38, -71.418, 30.555, 112.817, 12.894]
  MoveL 1865 to (227.28, 35.68, 41.04) mm, rotated rx -180 ry 0 rz 180 deg; joints [-27.942, 45.38, -71.418, 30.555, 112.817, 12.894]
  Call Extruder(191.82028)
  MoveL 1866 to (227.52, 35.73, 41.03) mm, rotated rx -180 ry 0 rz 180 deg; joints [-27.888, 45.404, -71.418, 30.492, 112.808, 12.859]
  MoveL 1867 to (227.52, 35.73, 41.03) mm, rotated rx -180 ry 0 rz 180 deg; joints [-27.888, 45.404, -71.418, 30.492, 112.808, 12.859]
  Call Extruder(191.95543)
  MoveL 1868 to (227.77, 35.78, 41.03) mm, rotated rx -180 ry 0 rz 180 deg; joints [-27.834, 45.428, -71.417, 30.43, 112.8, 12.823]
  MoveL 1869 to (227.77, 35.78, 41.03) mm, rotated rx -180 ry 0 rz 180 deg; joints [-27.834, 45.428, -71.417, 30.43, 112.8, 12.823]
  Call Extruder(192.09119)
  MoveL 1870 to (228.02, 35.83, 41.04) mm, rotated rx -180 ry 0 rz 180 deg; joints [-27.78, 45.452, -71.417, 30.367, 112.791, 12.788]
  MoveL 1871 to (228.02, 35.83, 41.04) mm, rotated rx -180 ry 0 rz 180 deg; joints [-27.78, 45.452, -71.417, 30.367, 112.791, 12.788]
  Call Extruder(192.22756)
  MoveL 1872 to (228.27, 35.88, 41.04) mm, rotated rx -180 ry 0 rz 180 deg; joints [-27.726, 45.475, -71.417, 30.306, 112.782, 12.753]
  MoveL 1873 to (228.27, 35.88, 41.04) mm, rotated rx -180 ry 0 rz 180 deg; joints [-27.726, 45.475, -71.417, 30.306, 112.782, 12.753]
  Call Extruder(192.36453)
  MoveL 1874 to (228.52, 35.93, 41.04) mm, rotated rx -180 ry 0 rz 180 deg; joints [-27.673, 45.499, -71.417, 30.244, 112.773, 12.718]
  MoveL 1875 to (228.52, 35.93, 41.04) mm, rotated rx -180 ry 0 rz 180 deg; joints [-27.673, 45.499, -71.417, 30.244, 112.773, 12.718]
  Call Extruder(192.50212)
  MoveL 1876 to (228.77, 35.98, 41.04) mm, rotated rx -180 ry 0 rz 180 deg; joints [-27.62, 45.523, -71.417, 30.183, 112.764, 12.683]
  MoveL 1877 to (228.77, 35.98, 41.04) mm, rotated rx -180 ry 0 rz 180 deg; joints [-27.62, 45.523, -71.417, 30.183, 112.764, 12.683]
  Call Extruder(192.61584)
  MoveL 1878 to (228.97, 36.03, 41.04) mm, rotated rx -180 ry 0 rz 180 deg; joints [-27.579, 45.543, -71.416, 30.135, 112.755, 12.655]
  MoveL 1879 to (228.97, 36.03, 41.04) mm, rotated rx -180 ry 0 rz 180 deg; joints [-27.579, 45.543, -71.416, 30.135, 112.755, 12.655]
  Call Extruder(192.73001)
  MoveL 1880 to (229.18, 36.07, 41.04) mm, rotated rx -180 ry 0 rz -180 deg; joints [-27.539, 45.563, -71.416, 30.089, 112.747, 12.628]
  MoveL 1881 to (229.18, 36.07, 41.04) mm, rotated rx -180 ry 0 rz -180 deg; joints [-27.539, 45.563, -71.416, 30.089, 112.747, 12.628]
  Call Extruder(192.84463)
  MoveL 1882 to (229.38, 36.12, 41.04) mm, rotated rx 180 ry 0 rz 180 deg; joints [-27.499, 45.583, -71.416, 30.042, 112.738, 12.601]
  MoveL 1883 to (229.38, 36.12, 41.04) mm, rotated rx 180 ry 0 rz 180 deg; joints [-27.499, 45.583, -71.416, 30.042, 112.738, 12.601]
  Call Extruder(192.95971)
  MoveL 1884 to (229.59, 36.16, 41.04) mm, rotated rx 180 ry 0 rz 180 deg; joints [-27.458, 45.602, -71.416, 29.995, 112.73, 12.573]
  MoveL 1885 to (229.59, 36.16, 41.04) mm, rotated rx 180 ry 0 rz 180 deg; joints [-27.458, 45.602, -71.416, 29.995, 112.73, 12.573]
  Call Extruder(193.08194)
  MoveL 1886 to (229.8, 36.22, 41.04) mm, rotated rx -180 ry 0 rz -180 deg; joints [-27.423, 45.623, -71.415, 29.953, 112.719, 12.547]
  MoveL 1887 to (229.8, 36.22, 41.04) mm, rotated rx -180 ry 0 rz -180 deg; joints [-27.423, 45.623, -71.415, 29.953, 112.719, 12.547]
  Call Extruder(193.21160)
  MoveL 1888 to (230.02, 36.28, 41.04) mm, rotated rx 180 ry 0 rz -180 deg; joints [-27.392, 45.646, -71.415, 29.915, 112.706, 12.522]
  MoveL 1889 to (230.02, 36.28, 41.04) mm, rotated rx 180 ry 0 rz -180 deg; joints [-27.392, 45.646, -71.415, 29.915, 112.706, 12.522]
  Call Extruder(193.34183)
  MoveL 1890 to (230.25, 36.35, 41.04) mm, rotated rx -180 ry 0 rz 180 deg; joints [-27.361, 45.668, -71.415, 29.878, 112.693, 12.497]
  MoveL 1891 to (230.25, 36.35, 41.04) mm, rotated rx -180 ry 0 rz 180 deg; joints [-27.361, 45.668, -71.415, 29.878, 112.693, 12.497]
  Call Extruder(193.47263)
  MoveL 1892 to (230.47, 36.42, 41.04) mm, rotated rx 180 ry 0 rz 180 deg; joints [-27.33, 45.691, -71.414, 29.84, 112.68, 12.472]
  MoveL 1893 to (230.47, 36.42, 41.04) mm, rotated rx 180 ry 0 rz 180 deg; joints [-27.33, 45.691, -71.414, 29.84, 112.68, 12.472]
  Call Extruder(193.60399)
  MoveL 1894 to (230.7, 36.49, 41.04) mm, rotated rx -180 ry 0 rz 180 deg; joints [-27.299, 45.713, -71.414, 29.803, 112.667, 12.447]
  MoveL 1895 to (230.7, 36.49, 41.04) mm, rotated rx -180 ry 0 rz 180 deg; joints [-27.299, 45.713, -71.414, 29.803, 112.667, 12.447]
  Call Extruder(193.72432)
  MoveL 1896 to (230.9, 36.55, 41.03) mm, rotated rx 180 ry 0 rz 180 deg; joints [-27.275, 45.734, -71.414, 29.773, 112.654, 12.426]
  MoveL 1897 to (230.9, 36.55, 41.03) mm, rotated rx 180 ry 0 rz 180 deg; joints [-27.275, 45.734, -71.414, 29.773, 112.654, 12.426]
  Call Extruder(193.84516)
  MoveL 1898 to (231.1, 36.62, 41.04) mm, rotated rx 180 ry 0 rz 180 deg; joints [-27.25, 45.754, -71.413, 29.743, 112.641, 12.405]
  MoveL 1899 to (231.1, 36.62, 41.04) mm, rotated rx 180 ry 0 rz 180 deg; joints [-27.25, 45.754, -71.413, 29.743, 112.641, 12.405]
  Call Extruder(193.96651)
  MoveL 1900 to (231.3, 36.68, 41.04) mm, rotated rx -180 ry 0 rz -180 deg; joints [-27.225, 45.775, -71.413, 29.712, 112.628, 12.383]
  MoveL 1901 to (231.3, 36.68, 41.04) mm, rotated rx -180 ry 0 rz -180 deg; joints [-27.225, 45.775, -71.413, 29.712, 112.628, 12.383]
  Call Extruder(194.08838)
  MoveL 1902 to (231.5, 36.75, 41.04) mm, rotated rx 180 ry 0 rz -180 deg; joints [-27.201, 45.795, -71.412, 29.682, 112.615, 12.362]
  MoveL 1903 to (231.5, 36.75, 41.04) mm, rotated rx 180 ry 0 rz -180 deg; joints [-27.201, 45.795, -71.412, 29.682, 112.615, 12.362]
  Call Extruder(194.21076)
  MoveL 1904 to (231.71, 36.82, 41.04) mm, rotated rx -180 ry 0 rz 180 deg; joints [-27.177, 45.816, -71.412, 29.652, 112.602, 12.341]
  MoveL 1905 to (231.71, 36.82, 41.04) mm, rotated rx -180 ry 0 rz 180 deg; joints [-27.177, 45.816, -71.412, 29.652, 112.602, 12.341]
  Call Extruder(194.33365)
  MoveL 1906 to (231.91, 36.88, 41.04) mm, rotated rx 180 ry 0 rz -180 deg; joints [-27.153, 45.836, -71.411, 29.623, 112.589, 12.32]
  MoveL 1907 to (231.91, 36.88, 41.04) mm, rotated rx 180 ry 0 rz -180 deg; joints [-27.153, 45.836, -71.411, 29.623, 112.589, 12.32]
  Call Extruder(194.51082)
  MoveL 1908 to (232.19, 37, 41.04) mm, rotated rx 180 ry 0 rz 180 deg; joints [-27.135, 45.866, -71.411, 29.598, 112.566, 12.297]
  MoveL 1909 to (232.19, 37, 41.04) mm, rotated rx 180 ry 0 rz 180 deg; joints [-27.135, 45.866, -71.411, 29.598, 112.566, 12.297]
  Call Extruder(194.72368)
  MoveL 1910 to (232.53, 37.15, 41.04) mm, rotated rx -180 ry 0 rz 180 deg; joints [-27.124, 45.902, -71.41, 29.579, 112.537, 12.273]
  MoveL 1911 to (232.53, 37.15, 41.04) mm, rotated rx -180 ry 0 rz 180 deg; joints [-27.124, 45.902, -71.41, 29.579, 112.537, 12.273]
  Call Extruder(194.91775)
  MoveL 1912 to (232.83, 37.29, 41.04) mm, rotated rx -180 ry 0 rz 180 deg; joints [-27.113, 45.934, -71.409, 29.56, 112.51, 12.251]
  MoveL 1913 to (232.83, 37.29, 41.04) mm, rotated rx -180 ry 0 rz 180 deg; joints [-27.113, 45.934, -71.409, 29.56, 112.51, 12.251]
  Call Extruder(195.11861)
  MoveL 1914 to (233.13, 37.45, 41.04) mm, rotated rx 180 ry 0 rz 180 deg; joints [-27.114, 45.967, -71.408, 29.554, 112.481, 12.233]
  MoveL 1915 to (233.13, 37.45, 41.04) mm, rotated rx 180 ry 0 rz 180 deg; joints [-27.114, 45.967, -71.408, 29.554, 112.481, 12.233]
  Call Extruder(195.32676)
  MoveL 1916 to (233.44, 37.62, 41.04) mm, rotated rx 180 ry 0 rz 180 deg; joints [-27.126, 46.002, -71.407, 29.559, 112.447, 12.219]
  MoveL 1917 to (233.44, 37.62, 41.04) mm, rotated rx 180 ry 0 rz 180 deg; joints [-27.126, 46.002, -71.407, 29.559, 112.447, 12.219]
  Call Extruder(195.53571)
  MoveL 1918 to (233.75, 37.8, 41.04) mm, rotated rx 180 ry 0 rz 180 deg; joints [-27.138, 46.036, -71.406, 29.565, 112.414, 12.205]
  MoveL 1919 to (233.75, 37.8, 41.04) mm, rotated rx 180 ry 0 rz 180 deg; joints [-27.138, 46.036, -71.406, 29.565, 112.414, 12.205]
  Call Extruder(195.74544)
  MoveL 1920 to (234.05, 37.98, 41.04) mm, rotated rx -180 ry 0 rz 180 deg; joints [-27.15, 46.07, -71.405, 29.571, 112.381, 12.191]
  MoveL 1921 to (234.05, 37.98, 41.04) mm, rotated rx -180 ry 0 rz 180 deg; joints [-27.15, 46.07, -71.405, 29.571, 112.381, 12.191]
  Call Extruder(195.86398)
  MoveL 1922 to (234.23, 38.08, 41.04) mm, rotated rx -180 ry 0 rz 180 deg; joints [-27.157, 46.089, -71.404, 29.574, 112.362, 12.183]
  MoveL 1923 to (234.23, 38.08, 41.04) mm, rotated rx -180 ry 0 rz 180 deg; joints [-27.157, 46.089, -71.404, 29.574, 112.362, 12.183]
  Call Extruder(196.19680)
  MoveL 1924 to (234.68, 38.4, 41.04) mm, rotated rx -180 ry 0 rz 180 deg; joints [-27.216, 46.143, -71.403, 29.625, 112.301, 12.177]
  MoveL 1925 to (234.68, 38.4, 41.04) mm, rotated rx -180 ry 0 rz 180 deg; joints [-27.216, 46.143, -71.403, 29.625, 112.301, 12.177]
  Call Extruder(196.53081)
  MoveL 1926 to (235.13, 38.73, 41.04) mm, rotated rx -180 ry 0 rz 180 deg; joints [-27.274, 46.196, -71.401, 29.675, 112.241, 12.171]
  MoveL 1927 to (235.13, 38.73, 41.04) mm, rotated rx -180 ry 0 rz 180 deg; joints [-27.274, 46.196, -71.401, 29.675, 112.241, 12.171]
  Call Extruder(196.69838)
  MoveL 1928 to (235.35, 38.9, 41.04) mm, rotated rx 180 ry 0 rz 180 deg; joints [-27.302, 46.223, -71.4, 29.699, 112.211, 12.168]
  Call Extruder(197.52772)
  MoveL 1929 to (236.39, 39.81, 41.04) mm, rotated rx -180 ry 0 rz 180 deg; joints [-27.525, 46.352, -71.394, 29.907, 112.047, 12.184]
  Call Extruder(198.15878)
  MoveL 1930 to (237.09, 40.6, 41.04) mm, rotated rx -180 ry 0 rz 180 deg; joints [-27.771, 46.447, -71.39, 30.147, 111.91, 12.228]
  MoveL 1931 to (237.09, 40.6, 41.04) mm, rotated rx -180 ry 0 rz 180 deg; joints [-27.771, 46.447, -71.39, 30.147, 111.91, 12.228]
  Call Extruder(198.35639)
  MoveL 1932 to (237.3, 40.85, 41.03) mm, rotated rx 180 ry 0 rz 180 deg; joints [-27.851, 46.476, -71.388, 30.225, 111.866, 12.242]
  Call Extruder(198.69040)
  MoveL 1933 to (237.63, 41.3, 41.04) mm, rotated rx -180 ry 0 rz 180 deg; joints [-28.012, 46.524, -71.386, 30.384, 111.788, 12.278]
  MoveL 1934 to (237.63, 41.3, 41.04) mm, rotated rx -180 ry 0 rz 180 deg; joints [-28.012, 46.524, -71.386, 30.384, 111.788, 12.278]
  Call Extruder(199.02322)
  MoveL 1935 to (237.96, 41.75, 41.04) mm, rotated rx -180 ry 0 rz 180 deg; joints [-28.17, 46.572, -71.384, 30.54, 111.711, 12.312]
  MoveL 1936 to (237.96, 41.75, 41.04) mm, rotated rx -180 ry 0 rz 180 deg; joints [-28.17, 46.572, -71.384, 30.54, 111.711, 12.312]
  Call Extruder(199.20245)
  MoveL 1937 to (238.13, 41.99, 41.04) mm, rotated rx -180 ry 0 rz 180 deg; joints [-28.256, 46.598, -71.382, 30.625, 111.669, 12.33]
  MoveL 1938 to (238.13, 41.99, 41.04) mm, rotated rx -180 ry 0 rz 180 deg; joints [-28.256, 46.598, -71.382, 30.625, 111.669, 12.33]
  Call Extruder(199.41057)
  MoveL 1939 to (238.31, 42.3, 41.04) mm, rotated rx 180 ry 0 rz 180 deg; joints [-28.375, 46.627, -71.381, 30.743, 111.618, 12.36]
  MoveL 1940 to (238.31, 42.3, 41.04) mm, rotated rx 180 ry 0 rz 180 deg; joints [-28.375, 46.627, -71.381, 30.743, 111.618, 12.36]
  Call Extruder(199.61791)
  MoveL 1941 to (238.49, 42.6, 41.04) mm, rotated rx 180 ry 0 rz 180 deg; joints [-28.493, 46.655, -71.379, 30.861, 111.567, 12.389]
  MoveL 1942 to (238.49, 42.6, 41.04) mm, rotated rx 180 ry 0 rz 180 deg; joints [-28.493, 46.655, -71.379, 30.861, 111.567, 12.389]
  Call Extruder(199.82447)
  MoveL 1943 to (238.66, 42.91, 41.04) mm, rotated rx 180 ry 0 rz 180 deg; joints [-28.61, 46.684, -71.377, 30.978, 111.516, 12.417]
  MoveL 1944 to (238.66, 42.91, 41.04) mm, rotated rx 180 ry 0 rz 180 deg; joints [-28.61, 46.684, -71.377, 30.978, 111.516, 12.417]
  Call Extruder(200.03025)
  MoveL 1945 to (238.84, 43.21, 41.04) mm, rotated rx -180 ry 0 rz 180 deg; joints [-28.727, 46.712, -71.376, 31.095, 111.464, 12.445]
  MoveL 1946 to (238.84, 43.21, 41.04) mm, rotated rx -180 ry 0 rz 180 deg; joints [-28.727, 46.712, -71.376, 31.095, 111.464, 12.445]
  Call Extruder(200.18856)
  MoveL 1947 to (238.94, 43.46, 41.04) mm, rotated rx 180 ry 0 rz 180 deg; joints [-28.834, 46.733, -71.374, 31.202, 111.423, 12.474]
  MoveL 1948 to (238.94, 43.46, 41.04) mm, rotated rx 180 ry 0 rz 180 deg; joints [-28.834, 46.733, -71.374, 31.202, 111.423, 12.474]
  Call Extruder(200.34626)
  MoveL 1949 to (239.05, 43.71, 41.04) mm, rotated rx -180 ry 0 rz 180 deg; joints [-28.939, 46.753, -71.373, 31.309, 111.382, 12.503]
  MoveL 1950 to (239.05, 43.71, 41.04) mm, rotated rx -180 ry 0 rz 180 deg; joints [-28.939, 46.753, -71.373, 31.309, 111.382, 12.503]
  Call Extruder(200.51634)
  MoveL 1951 to (239.16, 43.98, 41.04) mm, rotated rx -180 ry 0 rz 180 deg; joints [-29.054, 46.775, -71.372, 31.424, 111.337, 12.533]
  MoveL 1952 to (239.16, 43.98, 41.04) mm, rotated rx -180 ry 0 rz 180 deg; joints [-29.054, 46.775, -71.372, 31.424, 111.337, 12.533]
  Call Extruder(200.69866)
  MoveL 1953 to (239.29, 44.27, 41.04) mm, rotated rx 180 ry 0 rz 180 deg; joints [-29.178, 46.799, -71.37, 31.549, 111.288, 12.566]
  MoveL 1954 to (239.29, 44.27, 41.04) mm, rotated rx 180 ry 0 rz 180 deg; joints [-29.178, 46.799, -71.37, 31.549, 111.288, 12.566]
  Call Extruder(200.88022)
  MoveL 1955 to (239.41, 44.56, 41.04) mm, rotated rx -180 ry 0 rz 180 deg; joints [-29.301, 46.823, -71.369, 31.673, 111.24, 12.599]
  MoveL 1956 to (239.41, 44.56, 41.04) mm, rotated rx -180 ry 0 rz 180 deg; joints [-29.301, 46.823, -71.369, 31.673, 111.24, 12.599]
  Call Extruder(200.93707)
  MoveL 1957 to (239.44, 44.66, 41.04) mm, rotated rx -180 ry 0 rz 180 deg; joints [-29.343, 46.829, -71.368, 31.715, 111.225, 12.611]
  MoveL 1958 to (239.44, 44.66, 41.04) mm, rotated rx -180 ry 0 rz 180 deg; joints [-29.343, 46.829, -71.368, 31.715, 111.225, 12.611]
  Call Extruder(201.05031)
  MoveL 1959 to (239.5, 44.85, 41.03) mm, rotated rx 180 ry 0 rz 180 deg; joints [-29.428, 46.843, -71.367, 31.801, 111.194, 12.635]
  MoveL 1960 to (239.5, 44.85, 41.03) mm, rotated rx 180 ry 0 rz 180 deg; joints [-29.428, 46.843, -71.367, 31.801, 111.194, 12.635]
  Call Extruder(201.16311)
  MoveL 1961 to (239.56, 45.03, 41.04) mm, rotated rx -180 ry 0 rz 180 deg; joints [-29.512, 46.857, -71.367, 31.885, 111.163, 12.658]
  MoveL 1962 to (239.56, 45.03, 41.04) mm, rotated rx -180 ry 0 rz 180 deg; joints [-29.512, 46.857, -71.367, 31.885, 111.163, 12.658]
  Call Extruder(201.27546)
  MoveL 1963 to (239.62, 45.22, 41.04) mm, rotated rx 180 ry 0 rz 180 deg; joints [-29.596, 46.871, -71.366, 31.97, 111.132, 12.681]
  MoveL 1964 to (239.62, 45.22, 41.04) mm, rotated rx 180 ry 0 rz 180 deg; joints [-29.596, 46.871, -71.366, 31.97, 111.132, 12.681]
  Call Extruder(201.38737)
  MoveL 1965 to (239.68, 45.41, 41.04) mm, rotated rx 180 ry 0 rz -180 deg; joints [-29.679, 46.885, -71.365, 32.054, 111.101, 12.704]
  MoveL 1966 to (239.68, 45.41, 41.04) mm, rotated rx 180 ry 0 rz -180 deg; joints [-29.679, 46.885, -71.365, 32.054, 111.101, 12.704]
  Call Extruder(201.50878)
  MoveL 1967 to (239.75, 45.62, 41.04) mm, rotated rx 180 ry 0 rz 180 deg; joints [-29.77, 46.9, -71.364, 32.147, 111.067, 12.729]
  MoveL 1968 to (239.75, 45.62, 41.04) mm, rotated rx 180 ry 0 rz 180 deg; joints [-29.77, 46.9, -71.364, 32.147, 111.067, 12.729]
  Call Extruder(201.63957)
  MoveL 1969 to (239.82, 45.84, 41.03) mm, rotated rx 180 ry 0 rz 180 deg; joints [-29.871, 46.916, -71.363, 32.248, 111.03, 12.757]
  MoveL 1970 to (239.82, 45.84, 41.03) mm, rotated rx 180 ry 0 rz 180 deg; joints [-29.871, 46.916, -71.363, 32.248, 111.03, 12.757]
  Call Extruder(201.76979)
  MoveL 1971 to (239.88, 46.06, 41.04) mm, rotated rx -180 ry 0 rz 180 deg; joints [-29.97, 46.932, -71.362, 32.348, 110.994, 12.785]
  MoveL 1972 to (239.88, 46.06, 41.04) mm, rotated rx -180 ry 0 rz 180 deg; joints [-29.97, 46.932, -71.362, 32.348, 110.994, 12.785]
  Call Extruder(201.89946)
  MoveL 1973 to (239.95, 46.29, 41.04) mm, rotated rx -180 ry 0 rz 180 deg; joints [-30.069, 46.949, -71.36, 32.448, 110.957, 12.812]
  MoveL 1974 to (239.95, 46.29, 41.04) mm, rotated rx -180 ry 0 rz 180 deg; joints [-30.069, 46.949, -71.36, 32.448, 110.957, 12.812]
  Call Extruder(202.02855)
  MoveL 1975 to (240.02, 46.51, 41.04) mm, rotated rx -180 ry 0 rz 180 deg; joints [-30.168, 46.965, -71.359, 32.548, 110.921, 12.839]
  MoveL 1976 to (240.02, 46.51, 41.04) mm, rotated rx -180 ry 0 rz 180 deg; joints [-30.168, 46.965, -71.359, 32.548, 110.921, 12.839]
  Call Extruder(202.14360)
  MoveL 1977 to (240.06, 46.72, 41.04) mm, rotated rx 180 ry 0 rz 180 deg; joints [-30.263, 46.978, -71.358, 32.645, 110.887, 12.866]
  MoveL 1978 to (240.06, 46.72, 41.04) mm, rotated rx 180 ry 0 rz 180 deg; joints [-30.263, 46.978, -71.358, 32.645, 110.887, 12.866]
  Call Extruder(202.25820)
  MoveL 1979 to (240.11, 46.92, 41.04) mm, rotated rx 180 ry 0 rz 180 deg; joints [-30.358, 46.992, -71.357, 32.741, 110.854, 12.893]
  MoveL 1980 to (240.11, 46.92, 41.04) mm, rotated rx 180 ry 0 rz 180 deg; joints [-30.358, 46.992, -71.357, 32.741, 110.854, 12.893]
  Call Extruder(202.37235)
  MoveL 1981 to (240.15, 47.12, 41.04) mm, rotated rx 180 ry 0 rz 180 deg; joints [-30.453, 47.005, -71.356, 32.836, 110.821, 12.92]
  MoveL 1982 to (240.15, 47.12, 41.04) mm, rotated rx 180 ry 0 rz 180 deg; joints [-30.453, 47.005, -71.356, 32.836, 110.821, 12.92]
  Call Extruder(202.48605)
  MoveL 1983 to (240.2, 47.33, 41.04) mm, rotated rx -180 ry 0 rz 180 deg; joints [-30.548, 47.018, -71.355, 32.932, 110.788, 12.946]
  MoveL 1984 to (240.2, 47.33, 41.04) mm, rotated rx -180 ry 0 rz 180 deg; joints [-30.548, 47.018, -71.355, 32.932, 110.788, 12.946]
  Call Extruder(202.61146)
  MoveL 1985 to (240.24, 47.56, 41.04) mm, rotated rx 180 ry 0 rz 180 deg; joints [-30.653, 47.033, -71.354, 33.038, 110.751, 12.976]
  MoveL 1986 to (240.24, 47.56, 41.04) mm, rotated rx 180 ry 0 rz 180 deg; joints [-30.653, 47.033, -71.354, 33.038, 110.751, 12.976]
  Call Extruder(202.74844)
  MoveL 1987 to (240.29, 47.8, 41.03) mm, rotated rx 180 ry 0 rz 180 deg; joints [-30.768, 47.049, -71.353, 33.155, 110.71, 13.008]
  MoveL 1988 to (240.29, 47.8, 41.03) mm, rotated rx 180 ry 0 rz 180 deg; joints [-30.768, 47.049, -71.353, 33.155, 110.71, 13.008]
  Call Extruder(202.88480)
  MoveL 1989 to (240.34, 48.05, 41.04) mm, rotated rx 180 ry 0 rz 180 deg; joints [-30.884, 47.065, -71.352, 33.272, 110.67, 13.041]
  MoveL 1990 to (240.34, 48.05, 41.04) mm, rotated rx 180 ry 0 rz 180 deg; joints [-30.884, 47.065, -71.352, 33.272, 110.67, 13.041]
  Call Extruder(203.02056)
  MoveL 1991 to (240.39, 48.3, 41.03) mm, rotated rx 180 ry 0 rz 180 deg; joints [-30.999, 47.082, -71.351, 33.388, 110.629, 13.073]
  MoveL 1992 to (240.39, 48.3, 41.03) mm, rotated rx 180 ry 0 rz 180 deg; joints [-30.999, 47.082, -71.351, 33.388, 110.629, 13.073]
  Call Extruder(203.15571)
  MoveL 1993 to (240.44, 48.55, 41.04) mm, rotated rx -180 ry 0 rz 180 deg; joints [-31.114, 47.098, -71.349, 33.504, 110.589, 13.105]
  MoveL 1994 to (240.44, 48.55, 41.04) mm, rotated rx -180 ry 0 rz 180 deg; joints [-31.114, 47.098, -71.349, 33.504, 110.589, 13.105]
  Call Extruder(203.29025)
  MoveL 1995 to (240.49, 48.8, 41.04) mm, rotated rx -180 ry 0 rz -180 deg; joints [-31.228, 47.114, -71.348, 33.619, 110.548, 13.136]
  MoveL 1996 to (240.49, 48.8, 41.04) mm, rotated rx -180 ry 0 rz -180 deg; joints [-31.228, 47.114, -71.348, 33.619, 110.548, 13.136]
  Call Extruder(203.42417)
  MoveL 1997 to (240.54, 49.05, 41.04) mm, rotated rx -180 ry 0 rz 180 deg; joints [-31.342, 47.13, -71.347, 33.734, 110.508, 13.167]
  MoveL 1998 to (240.54, 49.05, 41.04) mm, rotated rx -180 ry 0 rz 180 deg; joints [-31.342, 47.13, -71.347, 33.734, 110.508, 13.167]
  Call Extruder(203.57204)
  MoveL 1999 to (240.59, 49.33, 41.04) mm, rotated rx -180 ry 0 rz 180 deg; joints [-31.47, 47.148, -71.346, 33.863, 110.463, 13.203]
